// TwinCAT 3 PLC project mas516_PLC
// ProgramVersion: 3.1.4023.0
// libraries:
//   Tc2_Standard, * (Beckhoff Automation GmbH)
//   Tc2_System, * (Beckhoff Automation GmbH)
//   Tc3_Module, * (Beckhoff Automation GmbH)
//   VisuDialogs, * (System)
// project tree:
//   / GlobalTextList.TcGTLO, MAIN.TcPOU, PlcTask.TcTTO, Visualization Manager.TcVMO (not stored)
//   HMI/Function blocks/ FB_ModifyAutomaticControlSettings.TcPOU
//   HMI/ G_Hmi.TcGVL, Main.TcVIS
//   HMI/Struct/ ST_ModifyAutomaticControlSettings.TcDUT
//   HMI/Sub/ Cylinder.TcVIS, Winch.TcVIS
//   Inputs/Function blocks/ FB_AnalogInputScaling.TcPOU, FB_Encoder.TcPOU, FB_JoystickInputScaling.TcPOU, FB_FlowMeterInputScaling.TcPOU
//   Inputs/Functions/ F_DegToRad.TcPOU
//   Inputs/ G_Inputs.TcGVL, G_Sensors.TcGVL, P_Inputs.TcPOU
//   Inputs/Struct/ ST_AnalogInput.TcDUT, ST_JoystickInputScaling.TcDUT, ST_AnalogInputStatus.TcDUT, ST_AnalogInputScaling.TcDUT, ST_FlowMeterInputScaling.TcDUT
//   Machine Control/Function blocks/ FB_CylController.TcPOU, FB_AutomaticControl.TcPOU, FB_AutomaticControlWinch.TcPOU, FB_ClosedLoopControl.TcPOU, FB_FeedforwardWinch.TcPOU, FB_MotionReferenceGenerator_limit.TcPOU, FB_OpenLoopControl.TcPOU, FB_OpenLoopControlWinch.TcPOU, FB_ResetIntegralController.TcPOU, FB_ValveOutputGenerator.TcPOU, FB_AutomaticControl_old.TcPOU, FB_Clock.TcPOU, FB_ManualControl.TcPOU, FB_FeedForwardCyl.TcPOU, GVL_1247965427.TcGVL, FB_RampGen.TcPOU, WinchAngle.TcPOU (not stored)
//   Machine Control/ G_HeightCorrection.TcGVL, G_Parameters.TcGVL, G_Work.TcGVL, P_MachineControl.TcPOU
//   Machine Control/Struct/ ST_AutomaticControlSettings.TcDUT, ST_ClosedLoopControlSettings.TcDUT, ST_MotionReferenceGeneratorSettings.TcDUT, ST_OpenLoopControlSettings.TcDUT, ST_Parameters.TcDUT, ST_ValveOutputGeneratorSettings.TcDUT
//   Outputs/Function blocks/ FB_ValveOutput.TcPOU
//   Outputs/ G_Outputs.TcGVL, P_Outputs.TcPOU
//   Outputs/Struct/ ST_ValveDeadBand.TcDUT, ST_ValveOutput.TcDUT
// real-time tasks:
//   TASK PlcTask: cycle T#1ms, priority 20, ADS port 350
// I/O:
//   DEVICE Device 3 (EtherCAT), AmsNetId 128.39.200.184.4.1
//     Term 1 (EK1100) [EK1100 EtherCAT Coupler (2A E-Bus)]
//       DI (EL1008) [EL1008 8Ch. Dig. Input 24V, 3ms]
//       Term 3 (EL2008) [EL2008 8Ch. Dig. Output 24V, 0.5A]
//       Term 4 (EL3068) [EL3068 8Ch. Ana. Input 0-10V]
//       Term 5 (EL3068) [EL3068 8Ch. Ana. Input 0-10V]
//       Term 6 (EL3174) [EL3174 4Ch. Ana. Input +/-10V Diff., +/-20mA SingleEnded, 16 Bit]
//       Term 7 (EL3255) [EL3255 5Ch. potentiometer measurement with sensor supply]
//       Term 8 (EL4104) [EL4104 4Ch. Ana. Output 0-10V, 16bit]
//       Term 9 (EL6751) [EL6751 CANopen Master]
//       Term 11 (EL9011) [EL9011 End Terminal]
//     Box 10 (Fraba EtherCAT) [Absolute Rotary Encoder IXARC V01.05]
//   DEVICE Device 1 (EL6751), AmsNetId 128.39.200.184.2.1
// variable links:
//   mas516_PLC/mas516_PLC Instance <-> Device 3 (EtherCAT)/Box 10 (Fraba EtherCAT)
//     PlcTask Inputs/G_Inputs.nEncoderValue <-> Encoder/Position Value
//   mas516_PLC/mas516_PLC Instance <-> Device 3 (EtherCAT)/Term 1 (EK1100)/DI (EL1008)
//     PlcTask Inputs/G_Inputs.bAutoModeSelector <-> Channel 2/Input
//     PlcTask Inputs/G_Inputs.bJoystickEnable <-> Channel 5/Input
//     PlcTask Inputs/G_Inputs.bManualModeSelector <-> Channel 1/Input
//     PlcTask Inputs/G_Inputs.bStartButton <-> Channel 3/Input
//     PlcTask Inputs/G_Inputs.bStopButton <-> Channel 4/Input
//   mas516_PLC/mas516_PLC Instance <-> Device 3 (EtherCAT)/Term 1 (EK1100)/Term 3 (EL2008)
//     PlcTask Outputs/G_Outputs.bGreenLight <-> Channel 1/Output
//     PlcTask Outputs/G_Outputs.bRedLight <-> Channel 2/Output
//     PlcTask Outputs/G_Outputs.stCylValveOutput.bEnable <-> Channel 4/Output
//     PlcTask Outputs/G_Outputs.stWinchValveOutput.bEnable <-> Channel 3/Output
//   mas516_PLC/mas516_PLC Instance <-> Device 3 (EtherCAT)/Term 1 (EK1100)/Term 4 (EL3068)
//     PlcTask Inputs/G_Inputs.stPressureCyl_A_PistonSide.nValue <-> AI Standard Channel 4/Value
//     PlcTask Inputs/G_Inputs.stPressureCyl_A_PistonSide.stStatus <-> AI Standard Channel 4/Status
//     PlcTask Inputs/G_Inputs.stPressureCyl_B_RodSide.nValue <-> AI Standard Channel 3/Value
//     PlcTask Inputs/G_Inputs.stPressureCyl_B_RodSide.stStatus <-> AI Standard Channel 3/Status
//     PlcTask Inputs/G_Inputs.stPressureReturn.nValue <-> AI Standard Channel 2/Value
//     PlcTask Inputs/G_Inputs.stPressureReturn.stStatus <-> AI Standard Channel 2/Status
//     PlcTask Inputs/G_Inputs.stPressureSupply.nValue <-> AI Standard Channel 1/Value
//     PlcTask Inputs/G_Inputs.stPressureSupply.stStatus <-> AI Standard Channel 1/Status
//     PlcTask Inputs/G_Inputs.stPressureWinch_A1_Input.nValue <-> AI Standard Channel 5/Value
//     PlcTask Inputs/G_Inputs.stPressureWinch_A1_Input.stStatus <-> AI Standard Channel 5/Status
//     PlcTask Inputs/G_Inputs.stPressureWinch_A_Input.nValue <-> AI Standard Channel 7/Value
//     PlcTask Inputs/G_Inputs.stPressureWinch_A_Input.stStatus <-> AI Standard Channel 7/Status
//     PlcTask Inputs/G_Inputs.stPressureWinch_B1_Output.nValue <-> AI Standard Channel 6/Value
//     PlcTask Inputs/G_Inputs.stPressureWinch_B1_Output.stStatus <-> AI Standard Channel 6/Status
//     PlcTask Inputs/G_Inputs.stPressureWinch_B_Output.nValue <-> AI Standard Channel 8/Value
//     PlcTask Inputs/G_Inputs.stPressureWinch_B_Output.stStatus <-> AI Standard Channel 8/Status
//   mas516_PLC/mas516_PLC Instance <-> Device 3 (EtherCAT)/Term 1 (EK1100)/Term 5 (EL3068)
//     PlcTask Inputs/G_Inputs.stPressureWinchDrain.nValue <-> AI Standard Channel 1/Value
//     PlcTask Inputs/G_Inputs.stPressureWinchDrain.stStatus <-> AI Standard Channel 1/Status
//   mas516_PLC/mas516_PLC Instance <-> Device 3 (EtherCAT)/Term 1 (EK1100)/Term 6 (EL3174)
//     PlcTask Inputs/G_Inputs.stFlowWinch.nValue <-> AI Standard Channel 1/Value
//     PlcTask Inputs/G_Inputs.stFlowWinch.stStatus <-> AI Standard Channel 1/Status
//   mas516_PLC/mas516_PLC Instance <-> Device 3 (EtherCAT)/Term 1 (EK1100)/Term 7 (EL3255)
//     PlcTask Inputs/G_Inputs.stJoyX.nValue <-> AI Standard Channel 2/Value
//     PlcTask Inputs/G_Inputs.stJoyX.stStatus <-> AI Standard Channel 2/Status
//     PlcTask Inputs/G_Inputs.stJoyY.nValue <-> AI Standard Channel 3/Value
//     PlcTask Inputs/G_Inputs.stJoyY.stStatus <-> AI Standard Channel 3/Status
//     PlcTask Inputs/G_Inputs.stPositionCylPiston.nValue <-> AI Standard Channel 1/Value
//     PlcTask Inputs/G_Inputs.stPositionCylPiston.stStatus <-> AI Standard Channel 1/Status
//   mas516_PLC/mas516_PLC Instance <-> Device 3 (EtherCAT)/Term 1 (EK1100)/Term 8 (EL4104)
//     PlcTask Outputs/G_Outputs.stCylValveOutput.nValveOutput <-> AO Output Channel 2/Analog output
//     PlcTask Outputs/G_Outputs.stWinchValveOutput.nValveOutput <-> AO Output Channel 1/Analog output

CONFIGURATION mas516_PLC
    RESOURCE PLC ON TwinCAT3
        TASK PlcTask(INTERVAL := T#1ms, PRIORITY := 20);
        PROGRAM MAIN WITH PlcTask : MAIN;
    END_RESOURCE
END_CONFIGURATION

// ---- HMI/Struct/ST_ModifyAutomaticControlSettings.TcDUT
TYPE ST_ModifyAutomaticControlSettings :
STRUCT
	bSetNewMaxFlowCapacity		: BOOL;
	fNewMaxFlowCapacity 		: LREAL;
	bSetNewProportionalGain 	: BOOL;
	bSetNewIntegralGain 		: BOOL;
	fNewProportionalGain 		: LREAL;
	fNewIntegralGain 			: LREAL;
	bSetNewMaxPositionError 	: BOOL;
	fNewMaxPositionError		: LREAL;
END_STRUCT
END_TYPE

// ---- Inputs/Struct/ST_AnalogInput.TcDUT
TYPE ST_AnalogInput :
STRUCT
	stStatus 	AT %I* : ST_AnalogInputStatus;
	nValue		AT %I* : INT;	
END_STRUCT
END_TYPE

// ---- Inputs/Struct/ST_JoystickInputScaling.TcDUT
TYPE ST_JoystickInputScaling :
STRUCT
	fMaxInputValue			: LREAL;	// tunable max input value
	fMinInputValue 			: LREAL;	// tunable min input value
	fNeutralInputValue  	: LREAL;	// tunable neutral input value
	fNeutralDeadband		: LREAL;	// tunable dead_band value
	fMaxOutputValue  		: LREAL;	// normalized max output value
	fMinOutputValue  		: LREAL;	// normalized min output value
	fNeutralOutputValue  	: LREAL;	// normalized neutral output value
END_STRUCT
END_TYPE

// ---- Inputs/Struct/ST_AnalogInputStatus.TcDUT
TYPE ST_AnalogInputStatus :
STRUCT
	Underrange 		: BIT; // 0.0
	Overrange 		: BIT; // 0.1
	Limit_1_0 		: BIT; // 0.2
	Limit_1_1 		: BIT; // 0.3
	Limit_2_0 		: BIT; // 0.4
	Limit_2_1 		: BIT; // 0.5
	Error 			: BIT; // 0.6
	Reserved_0_7	: BIT; // 0.7
	Reserved_1_0 	: BIT; // 1.0
	Reserved_1_1 	: BIT; // 1.1
	Reserved_1_2 	: BIT; // 1.2
	Reserved_1_3 	: BIT; // 1.3
	Reserved_1_4 	: BIT; // 1.4
	Reserved_1_5 	: BIT; // 1.5
	TxPDO_State 	: BIT; // 1.6
	TxPDO_Toggle 	: BIT; // 1.7	
END_STRUCT
END_TYPE

// ---- Inputs/Struct/ST_AnalogInputScaling.TcDUT
TYPE ST_AnalogInputScaling :
STRUCT
	fMaxInputValue 			: LREAL;	// tunable max input value 
	fMinInputValue			: LREAL;	// tunable min input value  
	fMaxOutputValue  		: LREAL;	// max sensor output value
	fMinOutputValue  		: LREAL;	// min sensor output value	
END_STRUCT
END_TYPE

// ---- Inputs/Struct/ST_FlowMeterInputScaling.TcDUT
TYPE ST_FlowMeterInputScaling :
STRUCT
	fMaxInputValue			: LREAL;	// tunable max input value
	fMinInputValue 			: LREAL;	// tunable min input value
	fNeutralInputValue  	: LREAL;	// tunable neutral input value
	fNeutralDeadband		: LREAL;	// tunable dead_band value
	fMaxOutputValue  		: LREAL;	// normalized max output value
	fMinOutputValue  		: LREAL;	// normalized min output value
	fNeutralOutputValue  	: LREAL;	// normalized neutral output value
END_STRUCT
END_TYPE

// ---- Machine Control/Struct/ST_AutomaticControlSettings.TcDUT
TYPE ST_AutomaticControlSettings :
STRUCT
	bEnableVelocityFeedForwardControl	: BOOL;
	bEnableClosedLoopPositionControl	: BOOL;
	bEnableIntegralController 			: BOOL;
	bEnableActiveDamping 				: BOOL;	
END_STRUCT
END_TYPE

// ---- Machine Control/Struct/ST_ClosedLoopControlSettings.TcDUT
TYPE ST_ClosedLoopControlSettings :
STRUCT
	fMaxPositionError 					: LREAL;
	fProportionalGain 					: LREAL;
	fIntegralGain 						: LREAL;
END_STRUCT
END_TYPE

// ---- Machine Control/Struct/ST_MotionReferenceGeneratorSettings.TcDUT
TYPE ST_MotionReferenceGeneratorSettings :
STRUCT
	fStartPosition_m		: LREAL := 0.0;
	fStartVelocity_m		: LREAL	:= 0.0;
	fPositionSetpoint_ms	: LREAL := 0.25;
	fVelocitySetpoint_m		: LREAL := 0.025;
	fMaxPosition 			: LREAL := 0.7;
	fMinPosition 			: LREAL := 0.0;
	fMaxVelocity 			: LREAL := 0.05;
	fTimeBeforeStarting_s	: LREAL := 3.0;
	fRampTime_s				: LREAL := 1.0;
	fHoldPositionTime_s		: LREAL := 5.0;
END_STRUCT
END_TYPE

// ---- Machine Control/Struct/ST_OpenLoopControlSettings.TcDUT
TYPE ST_OpenLoopControlSettings :
STRUCT
	fBoreArea 			: LREAL;
	fAnnulusArea 		: LREAL;
	fMaxFlowCapacity 	: LREAL; //[l/min]
END_STRUCT
END_TYPE

// ---- Machine Control/Struct/ST_Parameters.TcDUT
TYPE ST_Parameters :
STRUCT
	fCyclicTime 					: LREAL := 0.001; // [s]
	fMaxCylVelocityLimit 			: LREAL := 0.005; // [m/s]
	fMaxWinchVelocityLimit 			: LREAL := 0.005; // [rad/s]
	bDeadBandCompOn 				: BOOL := TRUE;
	stWinchValveDeadBand 			: ST_ValveDeadBand := (fPosMax := 29490.0, fPosMin := 20950.0, fNegMin := 18250.0, fNegMax := 9830.0);
	stCylValveDeadBand 				: ST_ValveDeadBand := (fPosMax := 29490.0, fPosMin := 20950.0, fNegMin := 18250.0, fNegMax := 9830.0);
	stPressureSensorScaling400bar 	: ST_AnalogInputScaling := (fMaxInputValue := 32767.0, fMinInputValue := 0.0, fMaxOutputValue := 400.0, fMinOutputValue := 0.0);
	stPressureSensorScaling40bar 	: ST_AnalogInputScaling := (fMaxInputValue := 32767.0, fMinInputValue := 0.0, fMaxOutputValue := 40.0, fMinOutputValue := 0.0);
	stJoystickInputScalingX 		: ST_JoystickInputScaling := (fMaxInputValue := 20509.0, fMinInputValue := 11787.0, fNeutralInputValue := 16175, fNeutralDeadband := 50.0, fMaxOutputValue := 1.0, fMinOutputValue := -1.0, fNeutralOutputValue := 0.0);
	stCylPistonPositionScaling 		: ST_AnalogInputScaling := (fMaxInputValue := 32295.0, fMinInputValue := 229.0, fMaxOutputValue := 0.5, fMinOutputValue := 0.0);
	stFlowMeterInputScaling 		: ST_FlowMeterInputScaling := (fMaxInputValue := 32295.0, fMinInputValue := 0.0, fNeutralInputValue := 15450, fNeutralDeadband := 50.0, fMaxOutputValue := 150.0, fMinOutputValue := -150.0, fNeutralOutputValue := 0.0);
	stJoystickInputScalingY 		: ST_JoystickInputScaling := (fMaxInputValue := 20504.0, fMinInputValue := 12160.0, fNeutralInputValue := 16640, fNeutralDeadband := 50.0, fMaxOutputValue := 1.0, fMinOutputValue := -1.0, fNeutralOutputValue := 0.0);
	fEncoderOffset 					: LREAL := 17574.8; // Encoder value at zero (Cylinder out / second layaer)
	fWinchDrumScaling				: LREAL := 0.000744309; //  (empirical value - combined drum diameter and gearing)
	fWinchSpeedReducerGain 			: LREAL := 0.2;
	fCylSpeedReducerGain 			: LREAL := 0.2;
	fDisplacment_cc 				: LREAL := 32;
	stWinchValveOutputGeneratorSettings  	: ST_ValveOutputGeneratorSettings := (fInitialValveOpening := 0.0, fValveOpeningSetPoint := 0.2, fTimeBeforeStarting_s := 3.0, fRampTime_s := 1.0, fHoldTime_s := 1.0, fWaitTime_s := 5.0);
	stCylValveOutputGeneratorSettings  		: ST_ValveOutputGeneratorSettings := (fInitialValveOpening := 0.0, fValveOpeningSetPoint := 0.2, fTimeBeforeStarting_s := 3.0, fRampTime_s := 1.0, fHoldTime_s := 1.0, fWaitTime_s := 5.0);
	stOpenLoopControlSettingsWinch 			: ST_OpenLoopControlSettings := (fBoreArea := 0.0, fAnnulusArea := 0.0, fMaxFlowCapacity := 60.0);
	stClosedLoopControlSettingsWinch 		: ST_ClosedLoopControlSettings := (fMaxPositionError := 2E-3, fProportionalGain := 9.7, fIntegralGain := 6.5);
	stOpenLoopControlSettingsCylinder 		: ST_OpenLoopControlSettings := (fBoreArea := 0.0033183, fAnnulusArea := 0.0023562, fMaxFlowCapacity := 75.0);
	stClosedLoopControlSettingsCylinder 	: ST_ClosedLoopControlSettings := (fMaxPositionError := 2E-3, fProportionalGain := 14.6, fIntegralGain := 9.75);	
END_STRUCT
END_TYPE

// ---- Machine Control/Struct/ST_ValveOutputGeneratorSettings.TcDUT
TYPE ST_ValveOutputGeneratorSettings :
STRUCT
	fInitialValveOpening	:	LREAL;
	fValveOpeningSetPoint	:	LREAL;
	fTimeBeforeStarting_s	:	LREAL;
	fRampTime_s				:	LREAL;
	fHoldTime_s				:	LREAL;
	fWaitTime_s				:	LREAL;
END_STRUCT
END_TYPE

// ---- Outputs/Struct/ST_ValveDeadBand.TcDUT
TYPE ST_ValveDeadBand :
STRUCT
	fPosMax	: LREAL; // Positive min value [19660..29490]
	fPosMin	: LREAL; // Positive max value [19660..29490]
	fNegMin : LREAL; // Negative max value [9830..19660]
	fNegMax	: LREAL; // Negative min value [9830..19660]
END_STRUCT
END_TYPE

// ---- Outputs/Struct/ST_ValveOutput.TcDUT
TYPE ST_ValveOutput :
STRUCT
	bEnable					AT %Q* : BOOL := 0;
	nValveOutput 			AT %Q* : INT := 19660;
END_STRUCT
END_TYPE

// ---- HMI/G_Hmi.TcGVL
{attribute 'qualified_only'}
VAR_GLOBAL
	bWinchEnable	: BOOL;
	bCylEnable 		: BOOL;
	stAutomaticControlSettingsWinch 			: ST_AutomaticControlSettings;
	stMotionReferenceGeneratorSettingsWinch  	: ST_MotionReferenceGeneratorSettings;
	stAutomaticControlSettingsCylinder 			: ST_AutomaticControlSettings;
	stMotionReferenceGeneratorSettingsCylinder  : ST_MotionReferenceGeneratorSettings;
	stModifyAutomaticControlSettingsWinch 		: ST_ModifyAutomaticControlSettings;
	stModifyAutomaticControlSettingsCylinder 	: ST_ModifyAutomaticControlSettings;
END_VAR

// ---- Inputs/G_Inputs.TcGVL
{attribute 'qualified_only'}
VAR_GLOBAL
	bManualModeSelector			AT %I* : BOOL;
	bAutoModeSelector			AT %I* : BOOL;
	bStartButton				AT %I* : BOOL;
	bStopButton					AT %I* : BOOL;
	bJoystickEnable				AT %I* : BOOL;
	
	// Analog Inputs 1
	stJoyX 						: ST_AnalogInput;
	stJoyY						: ST_AnalogInput;
	stPositionCylPiston 		: ST_AnalogInput;
	nEncoderValue 				AT %I* : UDINT;
	
	// Analog Inputs 2
	// HPU Interface
	stPressureSupply 			: ST_AnalogInput;
	stPressureReturn 			: ST_AnalogInput;
	// Cylinder
	stPressureCyl_A_PistonSide 	: ST_AnalogInput;
	stPressureCyl_B_RodSide		: ST_AnalogInput;
	// Winch
	stPressureWinch_A_Input 	: ST_AnalogInput;
	stPressureWinch_A1_Input 	: ST_AnalogInput;
	stPressureWinch_B_Output	: ST_AnalogInput;
	stPressureWinch_B1_Output	: ST_AnalogInput;
	stPressureWinchDrain		: ST_AnalogInput;
	
	// Analog Inputs 3 (Multi)
	stFlowWinch					: ST_AnalogInput;
END_VAR

// ---- Inputs/G_Sensors.TcGVL
{attribute 'qualified_only'}
VAR_GLOBAL
	fJoystickNormalizedY 		: LREAL;
	fJoystickNormalizedX 		: LREAL;
	fPositionCylPiston  		: LREAL;
	// HPU Interface
	fPressureSupply 			: LREAL;
	fPressureReturn 			: LREAL;
	// Cylinder
	fPressureCyl_A_PistonSide 	: LREAL;
	fPressureCyl_B_RodSide		: LREAL;
	// Winch
	fPressureWinch_A_Input 		: LREAL;
	fPressureWinch_A1_Side 		: LREAL;
	fPressureWinch_B_Output		: LREAL;
	fPressureWinch_B1_Output	: LREAL;
	fPressureWinchDrain			: LREAL;
	fWinchEncoderPosition 		: LREAL;
	fWinchWirePosition 			: LREAL;
	fWinchFlow 					: LREAL;	// [L/min]
END_VAR

// ---- Machine Control/Function blocks/GVL_1247965427.TcGVL
VAR_GLOBAL CONSTANT
	SS_INITIALIZE: SINT := 0;
	SS_STEP: SINT := 1;
END_VAR

// ---- Machine Control/G_HeightCorrection.TcGVL
{attribute 'qualified_only'}
VAR_GLOBAL
	xCorrectHeight : BOOL;
	rZeroOffset : REAL;
	rActual: REAL;
	rDesiredHeight: REAL;
END_VAR

// ---- Machine Control/G_Parameters.TcGVL
{attribute 'qualified_only'}
VAR_GLOBAL
	stParam : ST_Parameters;
END_VAR

// ---- Machine Control/G_Work.TcGVL
{attribute 'qualified_only'}
VAR_GLOBAL
	bManualMode 			: BOOL;
	bAutoMode 				: BOOL;
	bWinchEnable 			: BOOL;
	bCylEnable 				: BOOL;
	fWinchControlInput 		: LREAL;
	fWinchTime				: LREAL;
	fCylControlInput 		: LREAL;
	fCylTime				: LREAL;
	fVelRefWinch 			: LREAL;
	fPosRefWinch 			: LREAL;
	fControlSignWinch		: LREAL;
	fVelRefCyl 				: LREAL;
	fPosRefCyl 				: LREAL;
	fControlSignCyl			: LREAL;
	fPositionErrorWinch_mm 	: LREAL;
	fPositionErrorCylinder_mm : LREAL;
END_VAR

// ---- Outputs/G_Outputs.TcGVL
{attribute 'qualified_only'}
VAR_GLOBAL
	// PLC Rack
	
	// RIO Rack
	// Digital Outputs
	bGreenLight 			AT %Q* : BOOL;
	bRedLight 				AT %Q* : BOOL;
	// Analog Outputs
	stWinchValveOutput 		: ST_ValveOutput;
	stCylValveOutput 		: ST_ValveOutput;
END_VAR

// ---- MAIN.TcPOU
PROGRAM MAIN
VAR
END_VAR

P_Inputs();
P_MachineControl();
P_Outputs();

END_PROGRAM

// ---- Inputs/P_Inputs.TcPOU
PROGRAM P_Inputs
VAR
	fbJoystickWinch 				: FB_JoystickInputScaling;
	fbJoystickCyl 					: FB_JoystickInputScaling;
	fbWinchPosition 				: FB_Encoder;
	fbCylPistonPosition 			: FB_AnalogInputScaling;
	fbPressureSupply 				: FB_AnalogInputScaling;
	fbPressureReturn 				: FB_AnalogInputScaling;
	fbPressureCyl_A_PistonSide 		: FB_AnalogInputScaling;
	fbPressureCyl_B_RodSide			: FB_AnalogInputScaling;
	fbPressureWinch_A_Input 		: FB_AnalogInputScaling;
	fbPressureWinch_A1_Input 		: FB_AnalogInputScaling;
	fbPressureWinch_B_Output		: FB_AnalogInputScaling;
	fbPressureWinch_B1_Output		: FB_AnalogInputScaling;
	fbPressureWinchDrain			: FB_AnalogInputScaling;
	fbFlowWinch						: FB_FlowMeterInputScaling;
	
	
	
END_VAR

fbJoystickWinch(
	bEnable := G_Work.bManualMode,
	nRawInput := G_Inputs.stJoyY.nValue,
	stJoystickInputScaling := G_Parameters.stParam.stJoystickInputScalingY,
	fNormalizedOutput => G_Sensors.fJoystickNormalizedY
);

fbJoystickCyl(
	bEnable := G_Work.bManualMode,
	nRawInput := G_Inputs.stJoyX.nValue,
	stJoystickInputScaling := G_Parameters.stParam.stJoystickInputScalingX,
	fNormalizedOutput => G_Sensors.fJoystickNormalizedX
);

fbWinchPosition (
nRawInput := G_Inputs.nEncoderValue, 
fPosition => G_Sensors.fWinchEncoderPosition,
);

G_Sensors.fWinchWirePosition := fbWinchPosition.fPosition*G_Parameters.stParam.fWinchDrumScaling;

fbCylPistonPosition(
	nRawInput := G_Inputs.stPositionCylPiston.nValue,
	stAnalogInputScaling := G_Parameters.stParam.stCylPistonPositionScaling,
	fOutput => G_Sensors.fPositionCylPiston
);

fbPressureSupply(
	nRawInput := G_Inputs.stPressureSupply.nValue,
	stAnalogInputScaling := G_Parameters.stParam.stPressureSensorScaling400bar,
	fOutput => G_Sensors.fPressureSupply
);

fbPressureReturn(
	nRawInput := G_Inputs.stPressureReturn.nValue,
	stAnalogInputScaling := G_Parameters.stParam.stPressureSensorScaling40bar,
	fOutput => G_Sensors.fPressureReturn
);

fbPressureCyl_A_PistonSide(
	nRawInput := G_Inputs.stPressureCyl_A_PistonSide.nValue,
	stAnalogInputScaling := G_Parameters.stParam.stPressureSensorScaling400bar,
	fOutput => G_Sensors.fPressureCyl_A_PistonSide
);

fbPressureCyl_B_RodSide(
	nRawInput := G_Inputs.stPressureCyl_B_RodSide.nValue,
	stAnalogInputScaling := G_Parameters.stParam.stPressureSensorScaling400bar,
	fOutput => G_Sensors.fPressureCyl_B_RodSide
);

fbPressureWinch_A_Input(
	nRawInput := G_Inputs.stPressureWinch_A_Input.nValue,
	stAnalogInputScaling := G_Parameters.stParam.stPressureSensorScaling400bar,
	fOutput => G_Sensors.fPressureWinch_A_Input
);

fbPressureWinch_A1_Input(
	nRawInput := G_Inputs.stPressureWinch_A1_Input.nValue,
	stAnalogInputScaling := G_Parameters.stParam.stPressureSensorScaling400bar,
	fOutput => G_Sensors.fPressureWinch_A1_Side
);

fbPressureWinch_B_Output(
	nRawInput := G_Inputs.stPressureWinch_B_Output.nValue,
	stAnalogInputScaling := G_Parameters.stParam.stPressureSensorScaling400bar,
	fOutput => G_Sensors.fPressureWinch_B_Output
);

fbPressureWinch_B1_Output(
	nRawInput := G_Inputs.stPressureWinch_B1_Output.nValue,
	stAnalogInputScaling := G_Parameters.stParam.stPressureSensorScaling400bar,
	fOutput => G_Sensors.fPressureWinch_B1_Output
);

fbPressureWinchDrain(
	nRawInput := G_Inputs.stPressureWinchDrain.nValue,
	stAnalogInputScaling := G_Parameters.stParam.stPressureSensorScaling40bar,
	fOutput => G_Sensors.fPressureWinchDrain
);

fbFlowWinch(
	nRawInput := G_Inputs.stFlowWinch.nValue,
	stFlowMeterInputScaling := G_Parameters.stParam.stFlowMeterInputScaling,
	fNormalizedOutput => G_Sensors.fWinchFlow
);

END_PROGRAM

// ---- Inputs/Function blocks/FB_JoystickInputScaling.TcPOU
FUNCTION_BLOCK FB_JoystickInputScaling
VAR_INPUT
	bEnable 				: BOOL;
	nRawInput 				: INT;
	stJoystickInputScaling  : ST_JoystickInputScaling;
END_VAR
VAR_OUTPUT
	fNormalizedOutput 		: LREAL;
END_VAR
VAR
	fRawInput 				: LREAL;
	fTempInput 				: LREAL;
	fTempOutput 			: LREAL;
END_VAR

fRawInput := INT_TO_LREAL(nRawInput);

fTempInput := fRawInput - stJoystickInputScaling.fNeutralInputValue;

IF fTempInput > stJoystickInputScaling.fNeutralDeadband THEN
	fTempOutput := fTempInput/(stJoystickInputScaling.fMaxInputValue - stJoystickInputScaling.fNeutralInputValue);
ELSIF fTempInput < -stJoystickInputScaling.fNeutralDeadband THEN	
	fTempOutput := fTempInput/(stJoystickInputScaling.fNeutralInputValue - stJoystickInputScaling.fMinInputValue);
ELSE
	fTempOutput := 0.0;
END_IF

IF NOT(bEnable) THEN
	fNormalizedOutput := 0.0;
ELSE
	fNormalizedOutput := LIMIT(stJoystickInputScaling.fMinOutputValue, fTempOutput, stJoystickInputScaling.fMaxOutputValue);
END_IF

END_FUNCTION_BLOCK

// ---- Inputs/Function blocks/FB_Encoder.TcPOU
FUNCTION_BLOCK FB_Encoder
VAR_INPUT
	nRawInput : UDINT;
	stParam 		: ST_Parameters; 
END_VAR
VAR_OUTPUT
	fPosition 		: LREAL;
END_VAR
VAR PERSISTENT
	nRounds			: DINT;
	nRawLast 		: DINT;
END_VAR	
VAR
	nInput 		: DINT;
	nTempInputDiff	: DINT;
	nCount 			: DINT;
	nMaxValue30bit 	: DINT :=  1073741823; // 2^30 - 1	
	nThreshold30bit	: DINT := nMaxValue30bit/2;
	fScale16bit		: LREAL := 360.0/65535.0; // 360deg/(2^16 - 1)
	fTempPosition   : LREAL;
END_VAR

// Convert to DINT (same as const values)
nInput := UDINT_TO_DINT(nRawInput);

// Define Encoder Rounds
nTempInputDiff := nInput - nRawLast;
IF (nTempInputDiff > nThreshold30bit) THEN
	nRounds := nRounds - 1;
END_IF

IF (nTempInputDiff < -nThreshold30bit) THEN
	nRounds := nRounds + 1;
END_IF

// Count Encoder Rounds
nCount := nInput + nRounds*nMaxValue30bit;

//Position Output
fPosition := DINT_TO_LREAL(nCount)*fScale16bit - stParam.fEncoderOffset; // [deg]

END_FUNCTION_BLOCK

// ---- Inputs/Function blocks/FB_AnalogInputScaling.TcPOU
FUNCTION_BLOCK FB_AnalogInputScaling
VAR_INPUT
	nRawInput 				: INT;
	stAnalogInputScaling    : ST_AnalogInputScaling;
END_VAR
VAR_OUTPUT
	fOutput 				: LREAL;
END_VAR
VAR
	fRawInput 				: LREAL;
	fNormalizedInput		: LREAL;
END_VAR

fRawInput := INT_TO_LREAL(nRawInput);

fNormalizedInput := (fRawInput - stAnalogInputScaling.fMinInputValue) / (stAnalogInputScaling.fMaxInputValue - stAnalogInputScaling.fMinInputValue);

fOutput := LIMIT(stAnalogInputScaling.fMinOutputValue, stAnalogInputScaling.fMinOutputValue + fNormalizedInput*(stAnalogInputScaling.fMaxOutputValue - stAnalogInputScaling.fMinOutputValue), stAnalogInputScaling.fMaxOutputValue);

END_FUNCTION_BLOCK

// ---- Inputs/Function blocks/FB_FlowMeterInputScaling.TcPOU
FUNCTION_BLOCK FB_FlowMeterInputScaling
VAR_INPUT
	nRawInput 				: INT;
	stFlowMeterInputScaling  : ST_FlowMeterInputScaling;
END_VAR
VAR_OUTPUT
	fNormalizedOutput 		: LREAL;
END_VAR
VAR
	fRawInput 				: LREAL;
	fTempInput 				: LREAL;
	fTempOutput 			: LREAL;
END_VAR

fRawInput := INT_TO_LREAL(nRawInput);

fTempInput := fRawInput - stFlowMeterInputScaling.fNeutralInputValue;

IF fTempInput > stFlowMeterInputScaling.fNeutralDeadband THEN
	fTempOutput := fTempInput/(stFlowMeterInputScaling.fMaxInputValue - stFlowMeterInputScaling.fNeutralInputValue);
ELSIF fTempInput < -stFlowMeterInputScaling.fNeutralDeadband THEN	
	fTempOutput := fTempInput/(stFlowMeterInputScaling.fNeutralInputValue - stFlowMeterInputScaling.fMinInputValue);
ELSE
	fTempOutput := 0.0;
END_IF

fNormalizedOutput := LIMIT(stFlowMeterInputScaling.fMinOutputValue, fTempOutput*150.0, stFlowMeterInputScaling.fMaxOutputValue);

END_FUNCTION_BLOCK

// ---- Machine Control/P_MachineControl.TcPOU
PROGRAM P_MachineControl
VAR
	fbManualControlWinch 		: FB_ManualControl;
	fbManualControlCyl	 		: FB_ManualControl;
	//fbAutomaticControlWinch 	: FB_AutomaticControl_old;
	//fbAutomaticControlCyl	 	: FB_AutomaticControl_old;
	fWinchControlSignalManual 			: LREAL;
	fCylControlSignalManual 			: LREAL;
	fWinchControlSignalAuto 			: LREAL;
	fCylControlSignalAuto				: LREAL;
	fbAutomaticControlWinch 	:	FB_AutomaticControlWinch;
	fbAutomaticControlCylinder 		:	FB_AutomaticControl;
	fbModifyAutomaticControlSettingsWinch : FB_ModifyAutomaticControlSettings;
	fbModifyAutomaticControlSettingsCylinder : FB_ModifyAutomaticControlSettings;
END_VAR

G_Work.bManualMode := G_Inputs.bManualModeSelector;
G_Work.bAutoMode := G_Inputs.bAutoModeSelector;

G_Work.bWinchEnable := (G_Hmi.bWinchEnable AND G_Inputs.bJoystickEnable);
G_Work.bCylEnable :=  (G_Hmi.bCylEnable AND G_Inputs.bJoystickEnable);

fbManualControlWinch(
	bEnable := G_Work.bManualMode AND G_Work.bWinchEnable,
	fInput := G_Sensors.fJoystickNormalizedY*-G_Parameters.stParam.fWinchSpeedReducerGain,
	fControlRefSignal => fWinchControlSignalManual
);

fbManualControlCyl(
	bEnable := G_Work.bManualMode AND G_Work.bCylEnable,
	fInput := G_Sensors.fJoystickNormalizedX*G_Parameters.stParam.fCylSpeedReducerGain,
	fControlRefSignal => fCylControlSignalManual
);

//fbAutomaticControlWinch(
//	bEnable := G_Work.bAutoMode AND G_Hmi.bWinchEnable,
//	bStartMotion := G_Inputs.bStartButton,
//	bStopMotion := G_Inputs.bStopButton,
//	stValveOutputGeneratorSettings := G_Parameters.stWinchValveOutputGeneratorSettings,
//	fNormalizedValveOpeningRefSignal => fWinchControlSignalAuto,
//	fTime => G_Work.fWinchTime
//);

//fbAutomaticControlCyl(
//	bEnable := G_Work.bAutoMode AND G_Hmi.bCylEnable,
//	bStartMotion := G_Inputs.bStartButton,
//	bStopMotion := G_Inputs.bStopButton,
//	stValveOutputGeneratorSettings := G_Parameters.stCylValveOutputGeneratorSettings,
//	fNormalizedValveOpeningRefSignal => fCylControlSignalAuto,
//	fTime => G_Work.fCylTime
//);

fbModifyAutomaticControlSettingsWinch(
	stParamOpenLoopControllSettings := G_Parameters.stParam.stOpenLoopControlSettingsWinch,
	stParamClosedLoopControllSettings := G_Parameters.stParam.stClosedLoopControlSettingsWinch,	
	stModify := G_Hmi.stModifyAutomaticControlSettingsWinch
);

fbAutomaticControlWinch(
	bEnable := G_Work.bAutoMode AND G_Hmi.bWinchEnable,
	bStartMotion := G_Inputs.bStartButton,
	bStopMotion := G_Inputs.bStopButton,
	stMotionReferenceGeneratorSettings := G_Hmi.stMotionReferenceGeneratorSettingsWinch,
	stAutomaticControlSettings := G_Hmi.stAutomaticControlSettingsWinch,
	stClosedLoopControlSettings := G_Parameters.stParam.stClosedLoopControlSettingsWinch,
	stOpenLoopControlSettings := G_Parameters.stParam.stOpenLoopControlSettingsWinch,
	stParam := G_Parameters.stParam,
	fPositionFeedback := G_Sensors.fWinchWirePosition,
	fVelocityReference_ms => G_Work.fVelRefWinch,
	fPositionReference_m => G_Work.fPosRefWinch,
	fTime => G_Work.fWinchTime,
	fPositionError_mm => G_Work.fPositionErrorWinch_mm,
	fControlOutputNormalized => G_Work.fControlSignWinch
);


fbModifyAutomaticControlSettingsCylinder(
	stParamOpenLoopControllSettings := G_Parameters.stParam.stOpenLoopControlSettingsCylinder,
	stParamClosedLoopControllSettings := G_Parameters.stParam.stClosedLoopControlSettingsCylinder,	
	stModify := G_Hmi.stModifyAutomaticControlSettingsCylinder
);

fbAutomaticControlCylinder(
	bEnable := G_Work.bAutoMode AND G_Hmi.bCylEnable,
	bStartMotion := G_Inputs.bStartButton,
	bStopMotion := G_Inputs.bStopButton,
	stMotionReferenceGeneratorSettings := G_Hmi.stMotionReferenceGeneratorSettingsCylinder,
	stAutomaticControlSettings := G_Hmi.stAutomaticControlSettingsCylinder,
	stClosedLoopControlSettings := G_Parameters.stParam.stClosedLoopControlSettingsCylinder,
	stOpenLoopControlSettings := G_Parameters.stParam.stOpenLoopControlSettingsCylinder,
	stParam := G_Parameters.stParam,
	fPositionFeedback := G_Sensors.fPositionCylPiston,
	fVelocityReference_ms => G_Work.fVelRefCyl,
	fPositionReference_m => G_Work.fPosRefCyl,
	fTime => G_Work.fCylTime,
	fPositionError_mm => G_Work.fPositionErrorCylinder_mm,
	fControlOutputNormalized => G_Work.fControlSignCyl
);

IF G_Work.bManualMode THEN
	G_Work.fWinchControlInput := fWinchControlSignalManual;
	G_Work.fCylControlInput := fCylControlSignalManual;
ELSIF G_Work.bAutoMode THEN
	G_Work.fWinchControlInput := G_Work.fControlSignWinch;
	G_Work.fCylControlInput := -G_Work.fControlSignCyl;
ELSE
	G_Work.fWinchControlInput := 0.0; 
	G_Work.fCylControlInput := 0.0;
END_IF

END_PROGRAM

// ---- Machine Control/Function blocks/FB_ManualControl.TcPOU
FUNCTION_BLOCK FB_ManualControl
VAR_INPUT
	bEnable 			: BOOL;
	fInput 				: LREAL;
END_VAR
VAR_OUTPUT
	fControlRefSignal	: LREAL;
END_VAR
VAR
END_VAR

IF NOT(bEnable) THEN
	fControlRefSignal := 0.0;
ELSE
	fControlRefSignal := fInput;
END_IF

END_FUNCTION_BLOCK

// ---- Machine Control/Function blocks/FB_AutomaticControlWinch.TcPOU
FUNCTION_BLOCK FB_AutomaticControlWinch
VAR_INPUT
	bEnable 							: BOOL;
	bStartMotion 						: BOOL;
	bStopMotion 						: BOOL;
	stMotionReferenceGeneratorSettings  : ST_MotionReferenceGeneratorSettings;
	stAutomaticControlSettings 			: ST_AutomaticControlSettings;
	stClosedLoopControlSettings 		: ST_ClosedLoopControlSettings;
	stOpenLoopControlSettings			: ST_OpenLoopControlSettings;
	stParam 							: ST_Parameters; 
	fPositionFeedback					: LREAL;
	rWinchPosRad						: REAL;
	fbHeightCalc						: WinchAngle;
	rActPos								: REAL;
	rSetPos								: REAL;
END_VAR
VAR_OUTPUT
	fTime : LREAL;
	fVelocityReference_ms : LREAL;
	fPositionReference_m : LREAL;
	fControlOutputNormalized : LREAL;
	fPositionError_mm : LREAL;
END_VAR
VAR
	fbClock : FB_Clock;	
	fbMotionReferenceGenerator 		: FB_MotionReferenceGenerator_limit;	
	fbVelocityFeedForwardControl 	: FB_FeedForwardWinch;
	fbResetIntegralController 		: FB_ResetIntegralController; 
	fbClosedLoopPositionControl 	: FB_CylController;
END_VAR

fbClock(
	bEnable := bEnable,
	bStart := bStartMotion,
	bStop := bStopMotion,
	fCycleTime := G_Parameters.stParam.fCyclicTime
);

fbMotionReferenceGenerator(
	bEnable := bEnable,
	stMotionReferenceGeneratorSettings := stMotionReferenceGeneratorSettings,
	fClock_s := fbClock.fTime
);

fbVelocityFeedForwardControl(
	bEnable := stAutomaticControlSettings.bEnableVelocityFeedForwardControl,
	fInput_ms := fbMotionReferenceGenerator.fVelocityReference_ms,
	fDisplacment_cc := stParam.fDisplacment_cc,
	stOpenLoopControlSettings := stOpenLoopControlSettings,
	rCircumference := 0.07 * 3.14,
	rTransmission := 1.0
);

fbResetIntegralController(
	stClosedLoopControlSettings := stClosedLoopControlSettings,
	fPositionError_m := fbClosedLoopPositionControl.xCylErrormm,
	fVelocityReference_ms := fbMotionReferenceGenerator.fVelocityReference_ms
);

rWinchPosRad := 3.141 * G_Sensors.fWinchEncoderPosition / 180; 
fbHeightCalc(
	xCyl := G_Sensors.fPositionCylPiston,
	winchAngleRad :=rWinchPosRad,
	hZero := G_HeightCorrection.rZeroOffset,
	wheelHeight := 0.330,
	totalDistance := 1.451,
	spoolRadius := 0.04575);
	
G_HeightCorrection.rActual := fbHeightCalc.height;

IF G_HeightCorrection.xCorrectHeight=TRUE THEN
	rSetPos := G_HeightCorrection.rDesiredHeight;
	rActPos := G_HeightCorrection.rActual;
ELSE
	rSetPos := fbMotionReferenceGenerator.fPositionReference_m;
	rActPos := G_HeightCorrection.rActual;
END_IF


fbClosedLoopPositionControl(
	EnablePFC := stAutomaticControlSettings.bEnableClosedLoopPositionControl,
	PosRefm := rSetPos,
	VRefms := fbMotionReferenceGenerator.fVelocityReference_ms,
	PosFbm := rActPos,
	propGain := stClosedLoopControlSettings.fProportionalGain,
	integralGain := stClosedLoopControlSettings.fIntegralGain,
	maxPosError := stClosedLoopControlSettings.fMaxPositionError,
	EnableIntegral := stAutomaticControlSettings.bEnableIntegralController,
	ssMethodType := BOOL_TO_SINT(bEnable AND bStartMotion)
);

fVelocityReference_ms := fbMotionReferenceGenerator.fVelocityReference_ms;
fPositionReference_m := fbMotionReferenceGenerator.fPositionReference_m;
fTime := fbClock.fTime;
fPositionError_mm := fbClosedLoopPositionControl.xCylErrormm/1E3;

IF bEnable THEN
	fControlOutputNormalized := LIMIT(-1.0, (fbVelocityFeedForwardControl.fNormalizedOutput + fbClosedLoopPositionControl.SetValue), 1.0);
ELSE
	fControlOutputNormalized := 0.0;
END_IF

END_FUNCTION_BLOCK

// ---- Machine Control/Function blocks/FB_Clock.TcPOU
FUNCTION_BLOCK FB_Clock
VAR_INPUT
	bEnable 	: BOOL;
	bStart 		: BOOL;
	bStop 		: BOOL;
	fCycleTime  : LREAL;
END_VAR
VAR_OUTPUT
	fTime : LREAL;
END_VAR
VAR
END_VAR

IF bStart AND NOT(bStop) AND bEnable THEN
	fTime := fTime + fCycleTime;
ELSE
	fTime := 0.0;
END_IF

END_FUNCTION_BLOCK

// ---- Machine Control/Function blocks/FB_MotionReferenceGenerator_limit.TcPOU
FUNCTION_BLOCK FB_MotionReferenceGenerator_limit
VAR_INPUT
	bEnable 							: BOOL;
	stMotionReferenceGeneratorSettings  : ST_MotionReferenceGeneratorSettings;
	fClock_s							: LREAL;
END_VAR
VAR_OUTPUT
	fPositionReference_m	: LREAL;
	fVelocityReference_ms	: LREAL;
	fTotalMotionTime_s		: LREAL;
	bErrorSignal			: BOOL;
END_VAR
VAR
	fStartPosition_m		: LREAL;
	fStartVelocity_m		: LREAL;
	fPositionSetpoint_ms	: LREAL;
	fVelocitySetpoint_m		: LREAL;
	fTimeBeforeStarting_s	: LREAL;
	fRampTime_s				: LREAL;
	fHoldPositionTime_s		: LREAL;
	Error					: DINT;
	slopeExt				: LREAL;
	slopeRetr				: LREAL;
	tHold					: LREAL;
	x1						: LREAL;
	x4						: LREAL;
	x1_tmp					: LREAL;
	x1_tmp_tmp				: LREAL;
	x4_tmp					: LREAL;
	x4_tmp_tmp				: LREAL;
	x4_tmp_tmp_0			: LREAL;
	x1_tmp_0				: LREAL;
END_VAR

IF NOT(bEnable) THEN
	RETURN;
END_IF

// LIMIT function: https://help.codesys.com/api-content/2/codesys/3.5.12.0/en/_cds_operator_limit/
fStartPosition_m := LIMIT(stMotionReferenceGeneratorSettings.fMinPosition, stMotionReferenceGeneratorSettings.fStartPosition_m, stMotionReferenceGeneratorSettings.fMaxPosition);
fStartVelocity_m := LIMIT(0.0, stMotionReferenceGeneratorSettings.fStartVelocity_m, stMotionReferenceGeneratorSettings.fMaxVelocity);
fPositionSetpoint_ms := LIMIT(stMotionReferenceGeneratorSettings.fMinPosition, stMotionReferenceGeneratorSettings.fPositionSetpoint_ms, stMotionReferenceGeneratorSettings.fMaxPosition);
fVelocitySetpoint_m := LIMIT(0.0, stMotionReferenceGeneratorSettings.fVelocitySetpoint_m, stMotionReferenceGeneratorSettings.fMaxVelocity);
fTimeBeforeStarting_s := LIMIT(0.0, stMotionReferenceGeneratorSettings.fTimeBeforeStarting_s, 10.0);
fRampTime_s := LIMIT(0.0, stMotionReferenceGeneratorSettings.fRampTime_s, 10.0);
fHoldPositionTime_s := LIMIT(0.0, stMotionReferenceGeneratorSettings.fHoldPositionTime_s, 60.0);

slopeExt := fStartVelocity_m - fVelocitySetpoint_m;

slopeRetr := ( -fVelocitySetpoint_m) - fStartVelocity_m;

tHold := ((fPositionSetpoint_ms - fStartPosition_m) - (((fVelocitySetpoint_m * fVelocitySetpoint_m) - (fStartVelocity_m * fStartVelocity_m)) / (fVelocitySetpoint_m / fRampTime_s))) / fVelocitySetpoint_m;

IF tHold < 0.0  THEN 
    bErrorSignal := TRUE;
ELSE 
    bErrorSignal := FALSE;
END_IF;

x1_tmp_tmp := fTimeBeforeStarting_s + fRampTime_s;
x1_tmp := x1_tmp_tmp - fTimeBeforeStarting_s;
x1_tmp_0 := slopeExt / fRampTime_s;
x1 := ((x1_tmp * fStartVelocity_m) + fStartPosition_m) - ((x1_tmp_0 * (x1_tmp * x1_tmp)) / 2.0);

x4_tmp_tmp := x1_tmp_tmp + tHold;
x4_tmp_tmp_0 := x4_tmp_tmp + fRampTime_s;
x4_tmp := x4_tmp_tmp_0 + fHoldPositionTime_s;
x1_tmp := x4_tmp + fRampTime_s;
x4 := x1_tmp - x4_tmp;
x4 := (fPositionSetpoint_ms - (x4 * fStartVelocity_m)) + (((slopeRetr / fRampTime_s) * (x4 * x4)) / 2.0);

IF Error = 1 THEN 
    fPositionReference_m := fStartPosition_m;
    fVelocityReference_ms := fStartVelocity_m;
ELSIF (fClock_s >= 0.0) AND (fClock_s < fTimeBeforeStarting_s) THEN 
    fPositionReference_m := fStartPosition_m;
    fVelocityReference_ms := fStartVelocity_m;
ELSIF (fClock_s >= fTimeBeforeStarting_s) AND (fClock_s < x1_tmp_tmp) THEN 
    slopeRetr := fClock_s - fTimeBeforeStarting_s;
    fPositionReference_m := ((slopeRetr * fStartVelocity_m) + fStartPosition_m) - ((x1_tmp_0 * (slopeRetr * slopeRetr)) / 2.0);
    fVelocityReference_ms := fStartVelocity_m - (x1_tmp_0 * slopeRetr);
ELSIF (fClock_s >= x1_tmp_tmp) AND (fClock_s < x4_tmp_tmp) THEN 
    fPositionReference_m := ((fClock_s - x1_tmp_tmp) * fVelocitySetpoint_m) + x1;
    fVelocityReference_ms := fVelocitySetpoint_m;
ELSIF (fClock_s >= x4_tmp_tmp) AND (fClock_s < x4_tmp_tmp_0) THEN 
    slopeRetr := fClock_s - x4_tmp_tmp;
    fPositionReference_m := ((((x4_tmp_tmp - x1_tmp_tmp) * fVelocitySetpoint_m) + x1) + (slopeRetr * fVelocitySetpoint_m)) + ((x1_tmp_0 * (slopeRetr * slopeRetr)) / 2.0);
    fVelocityReference_ms := (slopeRetr * (slopeExt / fRampTime_s)) + fVelocitySetpoint_m;
ELSIF (fClock_s >= x4_tmp_tmp_0) AND (fClock_s < x4_tmp) THEN 
    fPositionReference_m := fPositionSetpoint_ms;
    fVelocityReference_ms := fStartVelocity_m;
ELSIF (fClock_s >= x4_tmp) AND (fClock_s < x1_tmp) THEN 
    slopeExt := fClock_s - x4_tmp;
    slopeRetr := slopeRetr / fRampTime_s;
    fPositionReference_m := (fPositionSetpoint_ms - (slopeExt * fStartVelocity_m)) + ((slopeRetr * (slopeExt * slopeExt)) / 2.0);
    fVelocityReference_ms := (slopeExt * slopeRetr) + fStartVelocity_m;
ELSE 
    x1_tmp_0 := x1_tmp + tHold;

    IF (fClock_s >= x1_tmp) AND (fClock_s < x1_tmp_0) THEN 
        fPositionReference_m := x4 - ((fClock_s - x1_tmp) * fVelocitySetpoint_m);
        fVelocityReference_ms :=  -fVelocitySetpoint_m;
    ELSIF (fClock_s >= x1_tmp_0) AND (fClock_s < (((((((fTimeBeforeStarting_s + fRampTime_s) + tHold) + fRampTime_s) + fHoldPositionTime_s) + fRampTime_s) + tHold) + fRampTime_s)) THEN 
        slopeExt := fClock_s - x1_tmp_0;
        slopeRetr := slopeRetr / fRampTime_s;
        fPositionReference_m := ((x4 - ((x1_tmp_0 - x1_tmp) * fVelocitySetpoint_m)) - (slopeExt * fVelocitySetpoint_m)) - ((slopeRetr * (slopeExt * slopeExt)) / 2.0);
        fVelocityReference_ms := ( -fVelocitySetpoint_m) - (slopeExt * slopeRetr);
    ELSE 
        fPositionReference_m := fStartPosition_m;
        fVelocityReference_ms := fStartVelocity_m;
    END_IF;

END_IF;

fTotalMotionTime_s := ((((((fTimeBeforeStarting_s + fRampTime_s) + tHold) + fRampTime_s) + fHoldPositionTime_s) + fRampTime_s) + tHold) + fRampTime_s;

END_FUNCTION_BLOCK

// ---- Machine Control/Function blocks/FB_FeedforwardWinch.TcPOU
FUNCTION_BLOCK FB_FeedforwardWinch
VAR_INPUT
	bEnable		: BOOL;
	fInput_ms	: LREAL;
	fDisplacment_cc : LREAL;
	rCircumference : REAL;
	stOpenLoopControlSettings : ST_OpenLoopControlSettings;
	rTransmission : REAL;
END_VAR
VAR_OUTPUT
	fNormalizedOutput: LREAL;
END_VAR
VAR
	fFlowReference_lmin : LREAL;
	fRads : LREAL;
END_VAR

fRads := fInput_ms * 3.14 * 2 * rTransmission / (rCircumference);
fFlowReference_lmin := (fDisplacment_cc*1E-5*fRads/(2*3.14))*60000;

IF bEnable THEN 
    fNormalizedOutput := (fFlowReference_lmin) / stOpenLoopControlSettings.fMaxFlowCapacity;
ELSE 
    fNormalizedOutput := 0.0;
END_IF;

IF fNormalizedOutput > 1.0 THEN
    fNormalizedOutput := 1.0;
ELSIF fNormalizedOutput < -1.0 THEN 
    fNormalizedOutput := -1.0;
END_IF;

END_FUNCTION_BLOCK

// ---- Machine Control/Function blocks/FB_ResetIntegralController.TcPOU
FUNCTION_BLOCK FB_ResetIntegralController
VAR_INPUT
	stClosedLoopControlSettings : ST_ClosedLoopControlSettings;
	fVelocityReference_ms	: LREAL;
	fPositionError_m		: LREAL;
END_VAR
VAR_OUTPUT
	bReset: BOOL;
END_VAR
VAR
END_VAR

IF ABS(fVelocityReference_ms) > 0.0 THEN 
    bReset := FALSE;
ELSIF ABS(fPositionError_m) > stClosedLoopControlSettings.fMaxPositionError THEN 
    bReset := FALSE;
ELSE 
    bReset := TRUE;
END_IF;

END_FUNCTION_BLOCK

// ---- Machine Control/Function blocks/FB_CylController.TcPOU
FUNCTION_BLOCK FB_CylController
VAR_INPUT
	ssMethodType: SINT;
	EnablePFC: BOOL;
	PosRefm: LREAL;
	PosFbm: LREAL;
	propGain: LREAL;
	vRefms: LREAL;
	integralGain: LREAL;
	EnableIntegral: BOOL;
	maxPosError: LREAL;
END_VAR
VAR_OUTPUT
	xCylErrormm: LREAL;
	SetValue: LREAL;
END_VAR
VAR
	rtb_Reset: LREAL;
	rtb_u_FB: LREAL;
	rtb_Saturation1: LREAL;
	c_DiscreteTimeIntegrator_DS: LREAL;
	Delay_DSTATE: ARRAY[0..1] OF LREAL;
END_VAR



CASE ssMethodType OF
    SS_INITIALIZE: 
        (* SystemInitialize for Atomic SubSystem: '<Root>/CylController' *)
        (* InitializeConditions for Delay: '<S1>/Delay' *)
        Delay_DSTATE[0] := 0.0;
        Delay_DSTATE[1] := 0.0;
        (* SystemInitialize for Atomic SubSystem: '<S1>/FB_ClosedLoopControl' *)
        (* InitializeConditions for DiscreteIntegrator: '<S2>/Discrete-Time Integrator' *)
        c_DiscreteTimeIntegrator_DS := 0.0;
        (* End of SystemInitialize for SubSystem: '<S1>/FB_ClosedLoopControl' *)
        (* End of SystemInitialize for SubSystem: '<Root>/CylController' *)
		SetValue := 0.0;
		c_DiscreteTimeIntegrator_DS := 0.0;
		PosRefm := 0.0;
		vRefms := 0.0;
    SS_STEP: 
        (* Outputs for Atomic SubSystem: '<Root>/CylController' *)
        (* Outputs for Atomic SubSystem: '<S1>/FB_ResetIntegralController' *)
        (* MATLAB Function: '<S3>/ResetIntegralController' *)
        (* MATLAB Function 'CylController/FB_ResetIntegralController/ResetIntegralController': '<S4>:1' *)
        (* '<S4>:1:3' if abs(vRef) > 0 || abs(exCyl) > exCylMax *)

        IF ABS(vRefms) > 0.0 THEN 
            ;
            ;
        ELSIF ABS(Delay_DSTATE[0]) > (0.001 * maxPosError) THEN 
            ;
            ;
        ELSE 
            (* Outputs for Atomic SubSystem: '<S1>/FB_ClosedLoopControl' *)
            (* DiscreteIntegrator: '<S2>/Discrete-Time Integrator' *)
            (* '<S4>:1:5' else *)
            (* '<S4>:1:6' Reset = 1; *)
            c_DiscreteTimeIntegrator_DS := 0.0;
            (* End of Outputs for SubSystem: '<S1>/FB_ClosedLoopControl' *)
        END_IF;

        (* End of MATLAB Function: '<S3>/ResetIntegralController' *)
        (* End of Outputs for SubSystem: '<S1>/FB_ResetIntegralController' *)
        

        (* Outputs for Atomic SubSystem: '<S1>/FB_ClosedLoopControl' *)
        (* DiscreteIntegrator: '<S2>/Discrete-Time Integrator' *)

        IF c_DiscreteTimeIntegrator_DS >= 1.0 THEN 
            c_DiscreteTimeIntegrator_DS := 1.0;
        ELSIF c_DiscreteTimeIntegrator_DS <= -1.0 THEN 
            c_DiscreteTimeIntegrator_DS := -1.0;
        END_IF;

        (* Sum: '<S2>/Sum1' *)
        rtb_Reset := PosRefm - PosFbm;
        (* Switch: '<S2>/Switch' incorporates:
         *  Constant: '<S2>/Constant'
         *  DiscreteIntegrator: '<S2>/Discrete-Time Integrator' *)

        IF EnableIntegral THEN 
            rtb_u_FB := c_DiscreteTimeIntegrator_DS;
        ELSE 
            rtb_u_FB := 0.0;
        END_IF;

        (* End of Switch: '<S2>/Switch' *)
        

        (* Sum: '<S2>/Sum5' incorporates:
         *  Product: '<S2>/Product' *)
        rtb_u_FB := (propGain * rtb_Reset) + rtb_u_FB;
        (* Saturate: '<S2>/Saturation1' *)

        IF rtb_u_FB > 1.0 THEN 
            rtb_Saturation1 := 1.0;
        ELSIF rtb_u_FB >= -1.0 THEN 
            rtb_Saturation1 := rtb_u_FB;
        ELSE 
            rtb_Saturation1 := -1.0;
        END_IF;

        (* End of Saturate: '<S2>/Saturation1' *)
        

        (* Switch: '<S2>/Switch1' *)

        IF EnablePFC THEN 
            (* Outport: '<Root>/Set Value' *)
            SetValue := rtb_Saturation1;
        ELSE 
            (* Outport: '<Root>/Set Value' incorporates:
             *  Constant: '<S2>/Constant1' *)
            SetValue := 0.0;
        END_IF;

        (* End of Switch: '<S2>/Switch1' *)
        

        (* Update for DiscreteIntegrator: '<S2>/Discrete-Time Integrator' incorporates:
         *  Product: '<S2>/Divide'
         *  Product: '<S2>/Product2'
         *  Sum: '<S2>/Sum2'
         *  Sum: '<S2>/Sum3' *)
        c_DiscreteTimeIntegrator_DS := (((((rtb_Saturation1 - rtb_u_FB) / propGain) + rtb_Reset) * integralGain) * 0.001) + c_DiscreteTimeIntegrator_DS;

        IF c_DiscreteTimeIntegrator_DS >= 1.0 THEN 
            c_DiscreteTimeIntegrator_DS := 1.0;
        ELSIF c_DiscreteTimeIntegrator_DS <= -1.0 THEN 
            c_DiscreteTimeIntegrator_DS := -1.0;
        END_IF;

        (* End of Update for DiscreteIntegrator: '<S2>/Discrete-Time Integrator' *)
        (* End of Outputs for SubSystem: '<S1>/FB_ClosedLoopControl' *)
        

        (* Update for Delay: '<S1>/Delay' *)
        Delay_DSTATE[0] := Delay_DSTATE[1];
        Delay_DSTATE[1] := rtb_Reset;
        (* Outport: '<Root>/xCylError [mm]' incorporates:
         *  Gain: '<S1>/Gain' *)
        xCylErrormm := 1000.0 * rtb_Reset;
        (* End of Outputs for SubSystem: '<Root>/CylController' *)
END_CASE;

END_FUNCTION_BLOCK

// ---- Machine Control/Function blocks/FB_AutomaticControl.TcPOU
FUNCTION_BLOCK FB_AutomaticControl
VAR_INPUT
	bEnable 							: BOOL;
	bStartMotion 						: BOOL;
	bStopMotion 						: BOOL;
	stMotionReferenceGeneratorSettings  : ST_MotionReferenceGeneratorSettings;
	stAutomaticControlSettings 			: ST_AutomaticControlSettings;
	stClosedLoopControlSettings 		: ST_ClosedLoopControlSettings;
	stOpenLoopControlSettings			: ST_OpenLoopControlSettings;
	stParam 							: ST_Parameters; 
	fPositionFeedback					: LREAL;
END_VAR
VAR_OUTPUT
	fTime : LREAL;
	fVelocityReference_ms : LREAL;
	fPositionReference_m : LREAL;
	fControlOutputNormalized : LREAL;
	fPositionError_mm : LREAL;
END_VAR
VAR
	fbClock : FB_Clock;	
	fbMotionReferenceGenerator 		: FB_MotionReferenceGenerator_limit;	
	fbVelocityFeedForwardControl 	: FB_FeedForwardCyl;
	fbResetIntegralController 		: FB_ResetIntegralController; 
	fbClosedLoopPositionControl 	: FB_CylController;
END_VAR

fbClock(
	bEnable := bEnable,
	bStart := bStartMotion,
	bStop := bStopMotion,
	fCycleTime := G_Parameters.stParam.fCyclicTime
);

fbMotionReferenceGenerator(
	bEnable := bEnable,
	stMotionReferenceGeneratorSettings := stMotionReferenceGeneratorSettings,
	fClock_s := fbClock.fTime
);

fbVelocityFeedForwardControl(
	Enable := stAutomaticControlSettings.bEnableVelocityFeedForwardControl,
	vRef_ms := fbMotionReferenceGenerator.fVelocityReference_ms,
	maxFlow_lmin := stOpenLoopControlSettings.fMaxFlowCapacity,
	cylOpeningForward := 0.00331,
	cylOpeningBackward := 0.00236,
);

(* fbResetIntegralController(
	stClosedLoopControlSettings := stClosedLoopControlSettings,
	fPositionError_m := fbClosedLoopPositionControl.fPositionError,
	fVelocityReference_ms := fbMotionReferenceGenerator.fVelocityReference_ms
);*)

(*fbClosedLoopPositionControl(
	bEnable := stAutomaticControlSettings.bEnableClosedLoopPositionControl,
	stParam := stParam,
	stClosedLoopControlSettings := stClosedLoopControlSettings,		
	bActivateIntegralController := stAutomaticControlSettings.bEnableIntegralController,
	bIntegralControllReset := fbResetIntegralController.bReset,
	fInput_m := fbMotionReferenceGenerator.fPositionReference_m,
	fFeedback_m := fPositionFeedback
);*)


fVelocityReference_ms := fbMotionReferenceGenerator.fVelocityReference_ms;
fPositionReference_m := fbMotionReferenceGenerator.fPositionReference_m;
fTime := fbClock.fTime;


fbClosedLoopPositionControl(
	EnablePFC := stAutomaticControlSettings.bEnableClosedLoopPositionControl,
	PosRefm := fbMotionReferenceGenerator.fPositionReference_m,
	VRefms := fbMotionReferenceGenerator.fVelocityReference_ms,
	PosFbm := fPositionFeedback,
	propGain := stClosedLoopControlSettings.fProportionalGain,
	integralGain := stClosedLoopControlSettings.fIntegralGain,
	maxPosError := stClosedLoopControlSettings.fMaxPositionError,
	EnableIntegral := stAutomaticControlSettings.bEnableIntegralController,
	ssMethodType := BOOL_TO_SINT(bEnable AND bStartMotion)
);

fPositionError_mm := fbClosedLoopPositionControl.xCylerrormm;

IF bEnable THEN
	fControlOutputNormalized := LIMIT(-1.0, (fbVelocityFeedForwardControl.FeedfowardOutput + fbClosedLoopPositionControl.SetValue), 1.0);
ELSE
	fControlOutputNormalized := 0.0;
END_IF

END_FUNCTION_BLOCK

// ---- Machine Control/Function blocks/FB_FeedForwardCyl.TcPOU
FUNCTION_BLOCK FB_FeedForwardCyl
VAR_INPUT
	Enable: BOOL;
	vRef_ms: LREAL;
	maxFlow_lmin: LREAL;
	cylOpeningForward: LREAL;
	cylOpeningBackward: LREAL;
END_VAR
VAR_OUTPUT
	FeedfowardOutput: LREAL;
END_VAR
VAR
	rtb_Switch: LREAL;
END_VAR


(* Outputs for Atomic SubSystem: '<Root>/FeedForward' *)
(* Switch: '<S1>/Switch1' *)

IF Enable THEN 
    (* Switch: '<S1>/Switch' incorporates:
     *  Constant: '<S1>/Constant'
     *  Product: '<S1>/Product1'
     *  Product: '<S1>/Product2'
     *  RelationalOperator: '<S1>/Relational Operator' *)

    IF vRef_ms >= 0.0 THEN 
        rtb_Switch := cylOpeningForward * vRef_ms;
    ELSE 
        rtb_Switch := vRef_ms * cylOpeningBackward;
    END_IF;

    (* End of Switch: '<S1>/Switch' *)
    

    (* Outport: '<Root>/FeedfowardOutput' incorporates:
     *  Constant: '<S1>/Constant2'
     *  Product: '<S1>/Divide'
     *  Product: '<S1>/Product' *)
    FeedfowardOutput := (60000.0 * rtb_Switch) / maxFlow_lmin;
ELSE 
    (* Outport: '<Root>/FeedfowardOutput' incorporates:
     *  Constant: '<S1>/Constant1' *)
    FeedfowardOutput := 0.0;
END_IF;

(* End of Switch: '<S1>/Switch1' *)
(* End of Outputs for SubSystem: '<Root>/FeedForward' *)

END_FUNCTION_BLOCK

// ---- HMI/Function blocks/FB_ModifyAutomaticControlSettings.TcPOU
FUNCTION_BLOCK FB_ModifyAutomaticControlSettings
VAR_INPUT
	stParamOpenLoopControllSettings 	: REFERENCE TO ST_OpenLoopControlSettings;
	stParamClosedLoopControllSettings 	: REFERENCE TO ST_ClosedLoopControlSettings;
	stModify 							: ST_ModifyAutomaticControlSettings;
END_VAR
VAR_OUTPUT
END_VAR
VAR
END_VAR

IF stModify.bSetNewMaxFlowCapacity THEN
	stParamOpenLoopControllSettings.fMaxFlowCapacity := stModify.fNewMaxFlowCapacity;
	stModify.bSetNewMaxFlowCapacity := FALSE;
END_IF

IF stModify.bSetNewProportionalGain THEN
	stParamClosedLoopControllSettings.fProportionalGain := stModify.fNewProportionalGain;
	stModify.bSetNewProportionalGain := FALSE;
END_IF

IF stModify.bSetNewIntegralGain THEN
	stParamClosedLoopControllSettings.fIntegralGain := stModify.fNewIntegralGain;
	stModify.bSetNewIntegralGain := FALSE;
END_IF

IF stModify.bSetNewMaxPositionError THEN
	stParamClosedLoopControllSettings.fMaxPositionError:= stModify.fNewMaxPositionError;
	stModify.bSetNewMaxPositionError := FALSE;
END_IF

END_FUNCTION_BLOCK

// ---- Outputs/P_Outputs.TcPOU
PROGRAM P_Outputs
VAR
	fbWinchValveOutput 		: FB_ValveOutput;
	fbCylValveOutput 		: FB_ValveOutput;
END_VAR

///////////////////// Winch //////////////////////////////
G_Outputs.stWinchValveOutput.bEnable := G_Work.bManualMode OR G_Work.bAutoMode; 

fbWinchValveOutput(
	bEnable := (G_Work.bWinchEnable OR G_Work.fWinchTime > 0.0) AND G_Hmi.bWinchEnable,
	bDeadBandCompOn := G_Parameters.stParam.bDeadBandCompOn,
	stValveDeadBand := G_Parameters.stParam.stWinchValveDeadBand,
	fNormalizedInput := G_Work.fWinchControlInput,
	nOutput => G_Outputs.stWinchValveOutput.nValveOutput
);

///////////////////// Cylinder //////////////////////////////
G_Outputs.stCylValveOutput.bEnable := G_Work.bManualMode OR G_Work.bAutoMode;

fbCylValveOutput(
	bEnable := (G_Work.bCylEnable OR G_Work.fCylTime > 0.0) AND G_Hmi.bCylEnable,
	bDeadBandCompOn := G_Parameters.stParam.bDeadBandCompOn,
	stValveDeadBand := G_Parameters.stParam.stCylValveDeadBand,
	fNormalizedInput := G_Work.fCylControlInput,
	nOutput => G_Outputs.stCylValveOutput.nValveOutput
);

END_PROGRAM

// ---- Outputs/Function blocks/FB_ValveOutput.TcPOU
FUNCTION_BLOCK FB_ValveOutput
VAR_INPUT
	bEnable 			: BOOL;
	bDeadBandCompOn 	: BOOL;
	stValveDeadBand 	: ST_ValveDeadBand;
	fNormalizedInput 	: LREAL;
END_VAR
VAR_OUTPUT
	bEnableValveOutput : BOOL;
	nOutput : INT; 
END_VAR
VAR
	nOffset 	: INT := 19660;
	nMaxValue	: INT := 29490;
	nMinValue 	: INT :=  9830;
	nTempOutput : INT;
END_VAR

IF	bDeadBandCompOn THEN
	IF fNormalizedInput > 0.0 THEN
		nTempOutput := LREAL_TO_INT(ABS(fNormalizedInput*(stValveDeadBand.fPosMax - stValveDeadBand.fPosMin) + stValveDeadBand.fPosMin));
	ELSIF fNormalizedInput < 0.0 THEN
		nTempOutput := LREAL_TO_INT(ABS(fNormalizedInput*(stValveDeadBand.fNegMax - stValveDeadBand.fNegMin) - stValveDeadBand.fNegMin));
	ELSE
		nTempOutput := nOffset;
	END_IF
ELSE
	IF fNormalizedInput > 0.0 THEN
		nTempOutput := LREAL_TO_INT(ABS(fNormalizedInput*(32767.0 - 19660.0) + 19660.0));
	ELSIF fNormalizedInput < 0.0 THEN
		nTempOutput := LREAL_TO_INT(ABS(fNormalizedInput*(0 - 19660.0) - 19660.0));
	ELSE
		nTempOutput := nOffset;
	END_IF	
END_IF	

IF bEnable THEN
	nOutput := LIMIT(nMinValue, nTempOutput, nMaxValue);
	bEnableValveOutput := TRUE; 
ELSE 	
	nOutput := nOffset;
	bEnableValveOutput := FALSE;	
END_IF

END_FUNCTION_BLOCK

// ---- Inputs/Functions/F_DegToRad.TcPOU
FUNCTION F_DegToRad : LREAL
VAR_INPUT
	fInputDeg 	: LREAL;
END_VAR
VAR
	fPi 		:LREAL := 3.14159265359;
END_VAR

F_DegToRad := fInputDeg*(fPi/180);

END_FUNCTION

// ---- Machine Control/Function blocks/FB_ClosedLoopControl.TcPOU
FUNCTION_BLOCK FB_ClosedLoopControl
VAR_INPUT
	bEnable						: BOOL;
	stParam 					: ST_Parameters; 
	stClosedLoopControlSettings : ST_ClosedLoopControlSettings;
	bActivateIntegralController	: BOOL;
	bIntegralControllReset		: BOOL;
	fInput_m					: LREAL;
	fFeedback_m					: LREAL;
END_VAR
VAR_OUTPUT
	fNormalizedOutput	: LREAL;
	fPositionError		: LREAL;
END_VAR
VAR
	rtb_u_FB					: LREAL;
	rtb_Saturation1				: LREAL;
	c_DiscreteTimeIntegrator_DS	: LREAL;
END_VAR

fPositionError := fInput_m - fFeedback_m;

IF bIntegralControllReset THEN 
	c_DiscreteTimeIntegrator_DS := 0.0;
END_IF;

IF c_DiscreteTimeIntegrator_DS >= 1.0 THEN 
	c_DiscreteTimeIntegrator_DS := 1.0;
ELSIF c_DiscreteTimeIntegrator_DS <= -1.0 THEN 
	c_DiscreteTimeIntegrator_DS := -1.0;
END_IF;

IF bActivateIntegralController THEN 
	rtb_u_FB := c_DiscreteTimeIntegrator_DS;
ELSE 
	rtb_u_FB := 0.0;
END_IF;

rtb_u_FB := (stClosedLoopControlSettings.fProportionalGain * fPositionError) + rtb_u_FB;

IF rtb_u_FB > 1.0 THEN 
	rtb_Saturation1 := 1.0;
ELSIF rtb_u_FB >= -1.0 THEN 
	rtb_Saturation1 := rtb_u_FB;
ELSE 
	rtb_Saturation1 := -1.0;
END_IF;

IF bEnable THEN 
	fNormalizedOutput := rtb_Saturation1;
ELSE 
	fNormalizedOutput := 0.0;
END_IF;

c_DiscreteTimeIntegrator_DS := (((((rtb_Saturation1 - rtb_u_FB) / stClosedLoopControlSettings.fProportionalGain) + fPositionError) * stClosedLoopControlSettings.fIntegralGain) * stParam.fCyclicTime) + c_DiscreteTimeIntegrator_DS;

IF c_DiscreteTimeIntegrator_DS >= 1.0 THEN 
	c_DiscreteTimeIntegrator_DS := 1.0;
ELSIF c_DiscreteTimeIntegrator_DS <= -1.0 THEN 
	c_DiscreteTimeIntegrator_DS := -1.0;
END_IF;

END_FUNCTION_BLOCK

// ---- Machine Control/Function blocks/FB_OpenLoopControl.TcPOU
FUNCTION_BLOCK FB_OpenLoopControl
VAR_INPUT
	bEnable		: BOOL;
	fInput_ms	: LREAL;
	stOpenLoopControlSettings : ST_OpenLoopControlSettings;
END_VAR
VAR_OUTPUT
	fNormalizedOutput: LREAL;
END_VAR
VAR
	fFlowReference_m3s : LREAL;
	fM3sToLmin : LREAL := 60000;
END_VAR

IF fInput_ms >= 0.0 THEN 
    fFlowReference_m3s := stOpenLoopControlSettings.fBoreArea * fInput_ms;
ELSE 
    fFlowReference_m3s := fInput_ms * stOpenLoopControlSettings.fAnnulusArea;
END_IF;

IF bEnable THEN 
    fNormalizedOutput := (fM3sToLmin * fFlowReference_m3s) / stOpenLoopControlSettings.fMaxFlowCapacity;
ELSE 
    fNormalizedOutput := 0.0;
END_IF;

IF fNormalizedOutput > 1.0 THEN 
    fNormalizedOutput := 1.0;
ELSIF fNormalizedOutput < -1.0 THEN 
    fNormalizedOutput := -1.0;
END_IF;

END_FUNCTION_BLOCK

// ---- Machine Control/Function blocks/FB_OpenLoopControlWinch.TcPOU
FUNCTION_BLOCK FB_OpenLoopControlWinch
VAR_INPUT
	bEnable		: BOOL;
	fInput_ms	: LREAL;
	fDisplacment_cc : LREAL;
	fLin_m_ToRot_deg_Scaling : LREAL;
	stOpenLoopControlSettings : ST_OpenLoopControlSettings;
END_VAR
VAR_OUTPUT
	fNormalizedOutput: LREAL;
END_VAR
VAR
	fFlowReference_lmin : LREAL;
	fRads : LREAL;
END_VAR

fRads := (fInput_ms/fLin_m_ToRot_deg_Scaling)*3.14/180;
//fFlowReference_lmin := (fDisplacment_cc*(fRads/(2*3.14)*60))/1000;
fFlowReference_lmin := (fDisplacment_cc*1E-5*fRads/(2*3.14))*60000;

IF bEnable THEN 
    fNormalizedOutput := (fFlowReference_lmin) / stOpenLoopControlSettings.fMaxFlowCapacity;
ELSE 
    fNormalizedOutput := 0.0;
END_IF;

IF fNormalizedOutput > 1.0 THEN 
    fNormalizedOutput := 1.0;
ELSIF fNormalizedOutput < -1.0 THEN 
    fNormalizedOutput := -1.0;
END_IF;

END_FUNCTION_BLOCK

// ---- Machine Control/Function blocks/FB_ValveOutputGenerator.TcPOU
FUNCTION_BLOCK FB_ValveOutputGenerator
VAR_INPUT
	bEnable: BOOL;
	stValveOutputGeneratorSettings : ST_ValveOutputGeneratorSettings;
	fClock_s: LREAL;
END_VAR
VAR_OUTPUT
	fNormalizedValveOutputRef: LREAL;
	fTotalMotionTime_s: LREAL;
END_VAR
VAR
	fInitialValveOpening: LREAL;
	fValveOpeningSetPoint: LREAL;
	fTimeBeforeStarting_s: LREAL;
	fRampTime_s: LREAL;
	fHoldTime_s: LREAL;
	fWaitTime_s: LREAL;
	slopeExt: LREAL;
	slopeRetr: LREAL;
	Error: DINT;
	tmp: LREAL;
	temp1: LREAL;
END_VAR

fInitialValveOpening	:= stValveOutputGeneratorSettings.fInitialValveOpening;
fValveOpeningSetPoint	:= stValveOutputGeneratorSettings.fValveOpeningSetPoint;
fTimeBeforeStarting_s	:= stValveOutputGeneratorSettings.fTimeBeforeStarting_s;
fRampTime_s				:= stValveOutputGeneratorSettings.fRampTime_s;
fHoldTime_s				:= stValveOutputGeneratorSettings.fHoldTime_s;
fWaitTime_s				:= stValveOutputGeneratorSettings.fWaitTime_s;

(* Outputs for Atomic SubSystem: '<Root>/FB_AutomaticValveOutputGenerator' *)
(* Saturate: '<S1>/Saturation2' *)

IF fValveOpeningSetPoint > 1.0 THEN 
    fNormalizedValveOutputRef := 1.0;
ELSIF fValveOpeningSetPoint >= 0.0 THEN 
    fNormalizedValveOutputRef := fValveOpeningSetPoint;
ELSE 
    fNormalizedValveOutputRef := 0.0;
END_IF;

(* End of Saturate: '<S1>/Saturation2' *)


(* MATLAB Function: '<S1>/AutomaticValveOutputGenerator' *)
(* MATLAB Function 'FB_AutomaticValveOutputGenerator/AutomaticValveOutputGenerator': '<S2>:1' *)
(* '<S2>:1:2' us=u_ref; *)
(* '<S2>:1:3' slopeExt=u0-us; *)
slopeExt := fInitialValveOpening - fNormalizedValveOutputRef;
(* '<S2>:1:4' slopeRetr=-us-u0; *)
slopeRetr := ( -fNormalizedValveOutputRef) - fInitialValveOpening;
(* '<S2>:1:6' if tHold < 0 *)

IF fHoldTime_s < 0.0 THEN 
    (* '<S2>:1:7' Error = 1; *)
    Error := 1;
ELSE 
    (* '<S2>:1:8' else *)
    (* '<S2>:1:9' Error = 0; *)
    Error := 0;
END_IF;

(* '<S2>:1:12' t1=tRamp; *)
(* '<S2>:1:13' t2=tHold; *)
(* '<S2>:1:14' t3=tRamp; *)
(* '<S2>:1:15' t4=tWait; *)
(* '<S2>:1:16' t5=t1; *)
(* '<S2>:1:17' t6=t2; *)
(* '<S2>:1:18' t7=t3; *)
(* '<S2>:1:20' if Error == 1 *)

IF Error = 1 THEN 
    (* '<S2>:1:21' u = u0; *)
    fNormalizedValveOutputRef := fInitialValveOpening;
ELSIF (fClock_s >= 0.0) AND (fClock_s < fTimeBeforeStarting_s) THEN 
    (* '<S2>:1:22' elseif t>=0 && t<t0 *)
    (* '<S2>:1:23' u = u0; *)
    fNormalizedValveOutputRef := fInitialValveOpening;
ELSE 
    tmp := fTimeBeforeStarting_s + fRampTime_s;

    IF (fClock_s >= fTimeBeforeStarting_s) AND (fClock_s < tmp) THEN 
        (* '<S2>:1:24' elseif t>=t0 && t<(t0+t1) *)
        (* '<S2>:1:25' u = u0-(slopeExt/t1)*(t-t0); *)
        fNormalizedValveOutputRef := fInitialValveOpening - ((slopeExt / fRampTime_s) * (fClock_s - fTimeBeforeStarting_s));
    ELSE 
        temp1 := tmp + fHoldTime_s;

        IF (fClock_s < tmp) OR (fClock_s >= temp1) THEN 
            tmp := temp1 + fRampTime_s;

            IF (fClock_s >= temp1) AND (fClock_s < tmp) THEN 
                (* '<S2>:1:28' elseif t>=(t0+t1+t2) && t<(t0+t1+t2+t3) *)
                (* '<S2>:1:29' u = us+(slopeExt/t3)*(t-(t0+t1+t2)); *)
                fNormalizedValveOutputRef := ((fClock_s - temp1) * (slopeExt / fRampTime_s)) + fNormalizedValveOutputRef;
            ELSE 
                temp1 := tmp + fWaitTime_s;

                IF (fClock_s >= tmp) AND (fClock_s < temp1) THEN 
                    (* '<S2>:1:30' elseif t>=(t0+t1+t2+t3) && t<(t0+t1+t2+t3+t4) *)
                    (* '<S2>:1:31' u = u0; *)
                    fNormalizedValveOutputRef := fInitialValveOpening;
                ELSE 
                    tmp := temp1 + fRampTime_s;

                    IF (fClock_s >= temp1) AND (fClock_s < tmp) THEN 
                        (* '<S2>:1:32' elseif t>=(t0+t1+t2+t3+t4) && t<(t0+t1+t2+t3+t4+t5) *)
                        (* '<S2>:1:33' u = u0+(slopeRetr/t5)*(t-(t0+t1+t2+t3+t4)); *)
                        fNormalizedValveOutputRef := ((fClock_s - temp1) * (slopeRetr / fRampTime_s)) + fInitialValveOpening;
                    ELSE 
                        temp1 := tmp + fHoldTime_s;

                        IF (fClock_s >= tmp) AND (fClock_s < temp1) THEN 
                            (* '<S2>:1:34' elseif t>=(t0+t1+t2+t3+t4+t5) && t<(t0+t1+t2+t3+t4+t5+t6) *)
                            (* '<S2>:1:35' u = -us; *)
                            fNormalizedValveOutputRef :=  -fNormalizedValveOutputRef;
                        ELSIF (fClock_s >= temp1) AND (fClock_s < (temp1 + fRampTime_s)) THEN 
                            (* '<S2>:1:36' elseif t>=(t0+t1+t2+t3+t4+t5+t6) && t<(t0+t1+t2+t3+t4+t5+t6+t7) *)
                            (* '<S2>:1:37' u = -us-(slopeRetr/t3)*(t-(t0+t1+t2+t3+t4+t5+t6)); *)
                            fNormalizedValveOutputRef := ( -fNormalizedValveOutputRef) - ((fClock_s - temp1) * (slopeRetr / fRampTime_s));
                        ELSE 
                            (* '<S2>:1:38' else *)
                            (* '<S2>:1:39' u = u0; *)
                            fNormalizedValveOutputRef := fInitialValveOpening;
                        END_IF;

                    END_IF;

                END_IF;

            END_IF;

        END_IF;

    END_IF;

END_IF;

(* Switch: '<S1>/Switch' *)
(* '<S2>:1:42' T = t0+t1+t2+t3+t4+t5+t6+t7; *)

IF  NOT bEnable THEN 
    fNormalizedValveOutputRef := fInitialValveOpening;
END_IF;

(* End of Switch: '<S1>/Switch' *)


(* Saturate: '<S1>/Saturation' *)

IF fNormalizedValveOutputRef > 1.0 THEN 
    (* Outport: '<Root>/fNormalizedValveOutputRef' *)
    fNormalizedValveOutputRef := 1.0;
ELSIF fNormalizedValveOutputRef < -1.0 THEN 
    (* Outport: '<Root>/fNormalizedValveOutputRef' *)
    fNormalizedValveOutputRef := -1.0;
END_IF;

(* End of Saturate: '<S1>/Saturation' *)


(* Outport: '<Root>/fTotalMotionTime_s' incorporates:
 *  MATLAB Function: '<S1>/AutomaticValveOutputGenerator' *)
fTotalMotionTime_s := ((((((fTimeBeforeStarting_s + fRampTime_s) + fHoldTime_s) + fRampTime_s) + fWaitTime_s) + fRampTime_s) + fHoldTime_s) + fRampTime_s;
(* End of Outputs for SubSystem: '<Root>/FB_AutomaticValveOutputGenerator' *)

END_FUNCTION_BLOCK

// ---- Machine Control/Function blocks/FB_AutomaticControl_old.TcPOU
FUNCTION_BLOCK FB_AutomaticControl_old
VAR_INPUT
	bEnable								: BOOL;
	bStartMotion 						: BOOL;
	bStopMotion 						: BOOL;
	stValveOutputGeneratorSettings  	: ST_ValveOutputGeneratorSettings;
	stParam 		: ST_Parameters; 
END_VAR
VAR_OUTPUT
	fTime : LREAL;
	fNormalizedValveOpeningRefSignal : LREAL;
END_VAR
VAR
	fbClock 					: FB_Clock;	
	fbValveOutputGenerator 		: FB_ValveOutputGenerator;	
END_VAR

fbClock(
	bEnable := bEnable,
	bStart := bStartMotion,
	bStop := bStopMotion,
	fCycleTime := stParam.fCyclicTime
);

fbValveOutputGenerator(
	bEnable := bEnable,
	stValveOutputGeneratorSettings := stValveOutputGeneratorSettings,
	fClock_s := fbClock.fTime
);

fNormalizedValveOpeningRefSignal := fbValveOutputGenerator.fNormalizedValveOutputRef;
fTime := fbClock.fTime;

END_FUNCTION_BLOCK

// ---- Machine Control/Function blocks/FB_RampGen.TcPOU
FUNCTION_BLOCK FB_RampGen
VAR_INPUT
	ssMethodType: SINT;
	Enable: BOOL;
	x0m: LREAL;
	v0ms: LREAL;
	Position_SPm: LREAL;
	Velocity_SPms: LREAL;
	t0s: LREAL;
	tRamps: LREAL;
	tHoldPoss: LREAL;
	StartAuto: BOOL;
	StopAuto: BOOL;
END_VAR
VAR_OUTPUT
	PosRef: LREAL;
	VelRef: LREAL;
END_VAR
VAR
	Error: DINT;
	tHold: LREAL;
	x1: LREAL;
	x4: LREAL;
	rtb_Time: LREAL;
	rtb_Saturation3: LREAL;
	a_tmp: LREAL;
	a_tmp_tmp: LREAL;
	a_tmp_0: LREAL;
	a_tmp_tmp_0: LREAL;
	a_tmp_tmp_1: LREAL;
	a_tmp_tmp_2: LREAL;
	x1_tmp: LREAL;
	x4_tmp: LREAL;
	c_DiscreteTimeIntegrator_DS: LREAL;
END_VAR



CASE ssMethodType OF
    SS_INITIALIZE: 
        (* SystemInitialize for Atomic SubSystem: '<Root>/Subsystem' *)
        (* InitializeConditions for DiscreteIntegrator: '<S2>/Discrete-Time Integrator' *)
        c_DiscreteTimeIntegrator_DS := 0.0;
        (* End of SystemInitialize for SubSystem: '<Root>/Subsystem' *)
    SS_STEP: 
        (* Outputs for Atomic SubSystem: '<Root>/Subsystem' *)
        (* MATLAB Function: '<S2>/MATLAB Function' incorporates:
         *  DiscreteIntegrator: '<S2>/Discrete-Time Integrator' *)
        (* MATLAB Function 'Subsystem/MotionReferenceTime/MATLAB Function': '<S4>:1' *)
        (* '<S4>:1:3' if StartClock == 1 && ~StopClock *)

        IF StartAuto AND ( NOT StopAuto) THEN 
            (* '<S4>:1:4' Time = Clock; *)
            rtb_Time := c_DiscreteTimeIntegrator_DS;
        ELSE 
            (* '<S4>:1:5' else *)
            (* '<S4>:1:6' Time = 0.0; *)
            rtb_Time := 0.0;
        END_IF;

        (* End of MATLAB Function: '<S2>/MATLAB Function' *)
        

        (* Outputs for Atomic SubSystem: '<S1>/RampMotionProfileGenerator' *)
        (* Saturate: '<S3>/Saturation3' *)

        IF Position_SPm > 0.5 THEN 
            rtb_Saturation3 := 0.5;
        ELSIF Position_SPm >= 0.0 THEN 
            rtb_Saturation3 := Position_SPm;
        ELSE 
            rtb_Saturation3 := 0.0;
        END_IF;

        (* End of Saturate: '<S3>/Saturation3' *)
        

        (* Saturate: '<S3>/Saturation2' *)

        IF Velocity_SPms > 0.12 THEN 
            PosRef := 0.12;
        ELSIF Velocity_SPms >= 0.0 THEN 
            PosRef := Velocity_SPms;
        ELSE 
            PosRef := 0.0;
        END_IF;

        (* End of Saturate: '<S3>/Saturation2' *)
        

        (* MATLAB Function: '<S3>/RampSignal' *)
        (* MATLAB Function 'Subsystem/RampMotionProfileGenerator/RampSignal': '<S5>:1' *)
        (* '<S5>:1:2' x_SP = x_ref - x0; *)
        (* '<S5>:1:3' vs=v_ref; *)
        (* '<S5>:1:4' slopeExt=v0-vs; *)
        (* '<S5>:1:5' slopeRetr=-vs-v0; *)
        (* '<S5>:1:7' as = vs/tRamp; *)
        (* '<S5>:1:8' s_acc=(vs^2-v0^2)/as; *)
        (* '<S5>:1:10' tHold=(x_SP-s_acc)/vs; *)
        tHold := ((rtb_Saturation3 - x0m) - (((PosRef * PosRef) - (v0ms * v0ms)) / (PosRef / tRamps))) / PosRef;
        (* '<S5>:1:12' if tHold < 0 *)

        IF tHold < 0.0 THEN 
            (* '<S5>:1:13' Error = 1; *)
            Error := 1;
        ELSE 
            (* '<S5>:1:14' else *)
            (* '<S5>:1:15' Error = 0; *)
            Error := 0;
        END_IF;

        (* '<S5>:1:18' t1=tRamp; *)
        (* '<S5>:1:19' t2=tHold; *)
        (* '<S5>:1:20' t3=tRamp; *)
        (* '<S5>:1:21' t4=tWait; *)
        (* '<S5>:1:22' t5=t1; *)
        (* '<S5>:1:23' t6=t2; *)
        (* '<S5>:1:24' t7=t3; *)
        (* '<S5>:1:26' x1 = x0 + v0*((t0+t1)-t0)-(slopeExt/t1)*((t0+t1)-t0)^2/2; *)
        a_tmp_tmp := t0s + tRamps;
        a_tmp := a_tmp_tmp - t0s;
        x1_tmp := (v0ms - PosRef) / tRamps;
        x1 := ((a_tmp * v0ms) + x0m) - ((x1_tmp * (a_tmp * a_tmp)) / 2.0);
        (* '<S5>:1:27' x2 = x1 + vs*((t0+t1+t2)-(t0+t1)); *)
        (* '<S5>:1:28' x4 = x_ref - v0*((t0+t1+t2+t3+t4+t5)-(t0+t1+t2+t3+t4))+(slopeRetr/t5)*((t0+t1+t2+t3+t4+t5)-(t0+t1+t2+t3+t4))^2/2; *)
        a_tmp_tmp_0 := a_tmp_tmp + tHold;
        a_tmp_tmp_1 := a_tmp_tmp_0 + tRamps;
        a_tmp := a_tmp_tmp_1 + tHoldPoss;
        a_tmp_tmp_2 := a_tmp + tRamps;
        a_tmp_0 := a_tmp_tmp_2 - a_tmp;
        x4_tmp := (( -PosRef) - v0ms) / tRamps;
        x4 := (rtb_Saturation3 - (a_tmp_0 * v0ms)) + ((x4_tmp * (a_tmp_0 * a_tmp_0)) / 2.0);
        (* '<S5>:1:29' x5 = x4-vs*((t0+t1+t2+t3+t4+t5+t6)-(t0+t1+t2+t3+t4+t5)); *)
        (* '<S5>:1:31' if Error == 1 *)

        IF Error = 1 THEN 
            (* '<S5>:1:32' x = x0; *)
            rtb_Saturation3 := x0m;
            (* '<S5>:1:33' v = v0; *)
            PosRef := v0ms;
        ELSIF (rtb_Time >= 0.0) AND (rtb_Time < t0s) THEN 
            (* '<S5>:1:34' elseif t>=0 && t<t0 *)
            (* '<S5>:1:35' x = x0; *)
            rtb_Saturation3 := x0m;
            (* '<S5>:1:36' v = v0; *)
            PosRef := v0ms;
        ELSIF (rtb_Time >= t0s) AND (rtb_Time < a_tmp_tmp) THEN 
            (* '<S5>:1:37' elseif t>=t0 && t<(t0+t1) *)
            (* '<S5>:1:38' x = x0 + v0*(t-t0)-(slopeExt/t1)*(t-t0)^2/2; *)
            rtb_Time := rtb_Time - t0s;
            rtb_Saturation3 := ((rtb_Time * v0ms) + x0m) - ((x1_tmp * (rtb_Time * rtb_Time)) / 2.0);
            (* '<S5>:1:39' v = v0-(slopeExt/t1)*(t-t0); *)
            PosRef := v0ms - (x1_tmp * rtb_Time);
        ELSIF (rtb_Time >= a_tmp_tmp) AND (rtb_Time < a_tmp_tmp_0) THEN 
            (* '<S5>:1:40' elseif t>=(t0+t1) && t<(t0+t1+t2) *)
            (* '<S5>:1:41' x = x1 + vs*(t-(t0+t1)); *)
            rtb_Saturation3 := ((rtb_Time - a_tmp_tmp) * PosRef) + x1;
            (* '<S5>:1:42' v = vs; *)
        ELSIF (rtb_Time >= a_tmp_tmp_0) AND (rtb_Time < a_tmp_tmp_1) THEN 
            (* '<S5>:1:43' elseif t>=(t0+t1+t2) && t<(t0+t1+t2+t3) *)
            (* '<S5>:1:44' x = x2+vs*(t-(t0+t1+t2))+(slopeExt/t3)*(t-(t0+t1+t2))^2/2; *)
            rtb_Time := rtb_Time - a_tmp_tmp_0;
            rtb_Saturation3 := ((((a_tmp_tmp_0 - a_tmp_tmp) * PosRef) + x1) + (rtb_Time * PosRef)) + ((x1_tmp * (rtb_Time * rtb_Time)) / 2.0);
            (* '<S5>:1:45' v = vs+(slopeExt/t3)*(t-(t0+t1+t2)); *)
            PosRef := (rtb_Time * x1_tmp) + PosRef;
        ELSIF (rtb_Time >= a_tmp_tmp_1) AND (rtb_Time < a_tmp) THEN 
            (* '<S5>:1:46' elseif t>=(t0+t1+t2+t3) && t<(t0+t1+t2+t3+t4) *)
            (* '<S5>:1:47' x = x_ref; *)
            (* '<S5>:1:48' v = v0; *)
            PosRef := v0ms;
        ELSIF (rtb_Time >= a_tmp) AND (rtb_Time < a_tmp_tmp_2) THEN 
            (* '<S5>:1:49' elseif t>=(t0+t1+t2+t3+t4) && t<(t0+t1+t2+t3+t4+t5) *)
            (* '<S5>:1:50' x = x_ref - v0*(t-(t0+t1+t2+t3+t4))+(slopeRetr/t5)*(t-(t0+t1+t2+t3+t4))^2/2; *)
            a_tmp := rtb_Time - a_tmp;
            rtb_Saturation3 := (rtb_Saturation3 - (a_tmp * v0ms)) + ((x4_tmp * (a_tmp * a_tmp)) / 2.0);
            (* '<S5>:1:51' v = v0+(slopeRetr/t5)*(t-(t0+t1+t2+t3+t4)); *)
            PosRef := (a_tmp * x4_tmp) + v0ms;
        ELSE 
            rtb_Saturation3 := a_tmp_tmp_2 + tHold;

            IF (rtb_Time >= a_tmp_tmp_2) AND (rtb_Time < rtb_Saturation3) THEN 
                (* '<S5>:1:52' elseif t>=(t0+t1+t2+t3+t4+t5) && t<(t0+t1+t2+t3+t4+t5+t6) *)
                (* '<S5>:1:53' x = x4-vs*(t-(t0+t1+t2+t3+t4+t5)); *)
                rtb_Saturation3 := x4 - ((rtb_Time - a_tmp_tmp_2) * PosRef);
                (* '<S5>:1:54' v = -vs; *)
                PosRef :=  -PosRef;
            ELSIF (rtb_Time >= rtb_Saturation3) AND (rtb_Time < (rtb_Saturation3 + tRamps)) THEN 
                (* '<S5>:1:55' elseif t>=(t0+t1+t2+t3+t4+t5+t6) && t<(t0+t1+t2+t3+t4+t5+t6+t7) *)
                (* '<S5>:1:56' x = x5-vs*(t-(t0+t1+t2+t3+t4+t5+t6))-(slopeRetr/t3)*(t-(t0+t1+t2+t3+t4+t5+t6))^2/2; *)
                rtb_Time := rtb_Time - rtb_Saturation3;
                rtb_Saturation3 := ((x4 - ((rtb_Saturation3 - a_tmp_tmp_2) * PosRef)) - (rtb_Time * PosRef)) - ((x4_tmp * (rtb_Time * rtb_Time)) / 2.0);
                (* '<S5>:1:57' v = -vs-(slopeRetr/t3)*(t-(t0+t1+t2+t3+t4+t5+t6)); *)
                PosRef := ( -PosRef) - (rtb_Time * x4_tmp);
            ELSE 
                (* '<S5>:1:58' else *)
                (* '<S5>:1:59' x = x0; *)
                rtb_Saturation3 := x0m;
                (* '<S5>:1:60' v = v0; *)
                PosRef := v0ms;
            END_IF;

        END_IF;

        (* End of MATLAB Function: '<S3>/RampSignal' *)
        

        (* Switch: '<S3>/Switch' *)
        (* '<S5>:1:63' T = t0+t1+t2+t3+t4+t5+t6+t7; *)

        IF  NOT Enable THEN 
            PosRef := v0ms;
        END_IF;

        (* End of Switch: '<S3>/Switch' *)
        

        (* Saturate: '<S3>/Saturation' *)

        IF PosRef > 150.0 THEN 
            (* Outport: '<Root>/VelRef' *)
            VelRef := 150.0;
        ELSIF PosRef >= -150.0 THEN 
            (* Outport: '<Root>/VelRef' *)
            VelRef := PosRef;
        ELSE 
            (* Outport: '<Root>/VelRef' *)
            VelRef := -150.0;
        END_IF;

        (* End of Saturate: '<S3>/Saturation' *)
        

        (* Switch: '<S3>/Switch1' *)

        IF Enable THEN 
            PosRef := rtb_Saturation3;
        ELSE 
            PosRef := x0m;
        END_IF;

        (* End of Switch: '<S3>/Switch1' *)
        

        (* Saturate: '<S3>/Saturation1' *)

        IF PosRef > 500.0 THEN 
            (* Outport: '<Root>/PosRef' *)
            PosRef := 500.0;
        ELSIF PosRef < 0.0 THEN 
            (* Outport: '<Root>/PosRef' *)
            PosRef := 0.0;
        END_IF;

        (* End of Saturate: '<S3>/Saturation1' *)
        (* End of Outputs for SubSystem: '<S1>/RampMotionProfileGenerator' *)
        

        (* Update for DiscreteIntegrator: '<S2>/Discrete-Time Integrator' *)
        c_DiscreteTimeIntegrator_DS := c_DiscreteTimeIntegrator_DS + 0.001;
        (* End of Outputs for SubSystem: '<Root>/Subsystem' *)
END_CASE;

END_FUNCTION_BLOCK

// ---- GlobalTextList.TcGTLO
TEXTLIST GlobalTextList
  534 = 'Actual Height: %f'
  501 = 'Actual Height: %f [m]'
  920 = 'Closed Loop Position Control ON'
  583 = 'Current Cylinder Pos: %f [m] '
  824 = 'Current Drum Pos: %f [m] '
  35 = 'Current Drum Pos: %f [°] '
  829 = 'Current I-gain: %0.1f '
  196 = 'Current MaxError: %f [m] '
  955 = 'Current MaxFlow: %0.1f [L/min] '
  137 = 'Current P-gain: %0.1f '
  907 = 'Current Position: %f [m] '
  296 = 'Current Wire Pos: %f [m] '
  628 = 'Cylinder'
  783 = 'Desired Height: %f'
  51 = 'Desired Height: %f [m]'
  854 = 'Enable Cyl'
  32 = 'Enable Winch'
  995 = 'error: %f'
  246 = 'Error: %f [mm]'
  928 = 'Error: %f [m]'
  392 = 'Feed Forward Tuning'
  423 = 'Height stabilisation'
  252 = 'Height: %f'
  904 = 'Hold Pos time: %0.1f [s] '
  81 = 'Integral Controller Gain'
  573 = 'Integral Controller ON'
  261 = 'Max Position Error'
  415 = 'Motion Reference Generator Settings'
  655 = 'New I-gain: %0.1f '
  683 = 'New MaxError: %f  [m]'
  330 = 'New MaxFlow: %0.1f [L/min] '
  347 = 'New P-gain: %0.1f '
  463 = 'Position SP: %f [m] '
  982 = 'Proportional  Controller Gain'
  215 = 'Ramp time: %0.1f [s] '
  695 = 'Set New Value'
  828 = 'Start delay: %0.1f [s] '
  775 = 'Start Height: %f [m] '
  78 = 'Start Position: %f [m] '
  983 = 'Start Velocity: %f [m/s] '
  999 = 'Velocity SP: %f [m/s] '
  560 = 'VelocityFeed Forward Controller ON'
  349 = 'Winch'
  599 = 'Zero offset: %f '
  396 = 'Zero offset: %f [m]'
  522 = 'Zero offset: %f [m] '
END_TEXTLIST

// ---- HMI/Main.TcVIS
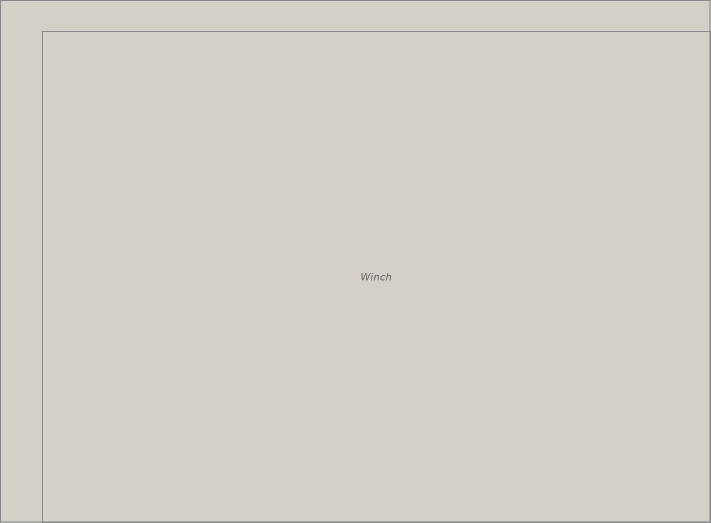
VISUALIZATION Main  // 711x523
    TabControl (42,31 669x492)
        shows Winch()
        shows Cylinder()
        [0]: TabTitle=Winch
        [1]: TabTitle=Cylinder
END_VISUALIZATION

// ---- HMI/Sub/Cylinder.TcVIS
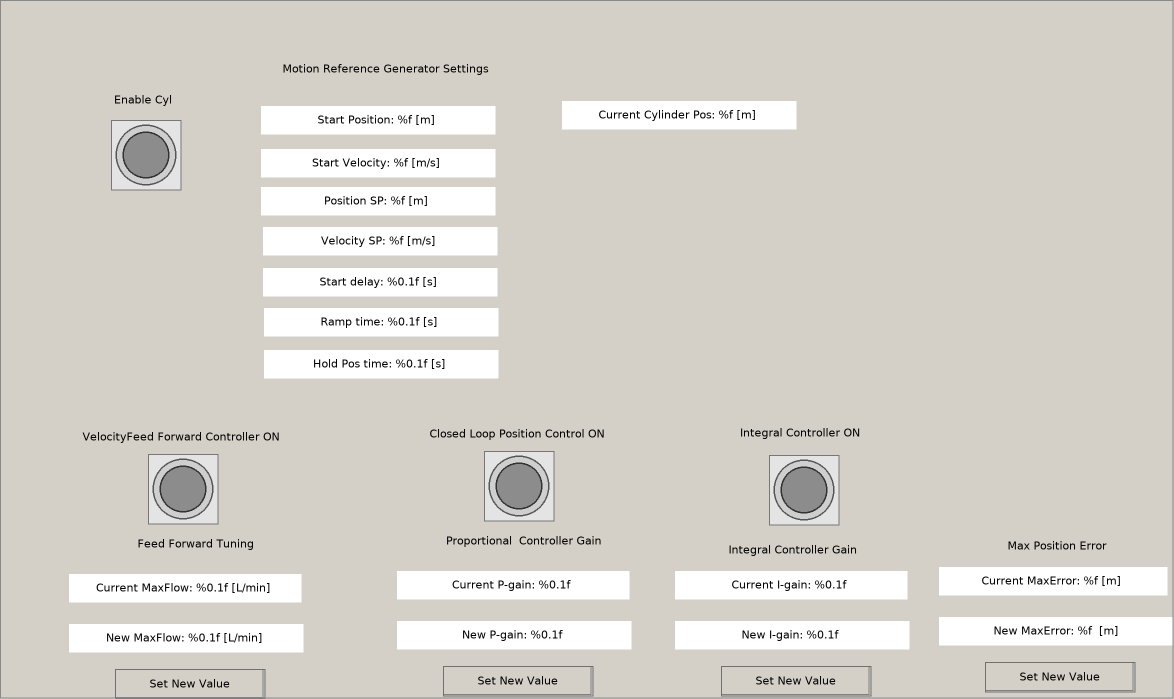
VISUALIZATION Cylinder  // 1174x699
    Label (68,85 150x30), "Enable Cyl"
    PushSwitch (111,120 70x70), variable: G_Hmi.bCylEnable, behaviour: TOGGLE, style: Switch-PushSwitch-Gray
    Label (240,54 291x30), "Motion Reference Generator Settings"
    Textfield (260,105 236x30), "Start Position: %f [m]", text variable: G_Hmi.stMotionReferenceGeneratorSettingsCylinder.fStartPosition_m
        OnMouseDown: write the text variable via Default, min 0, max 0.5
    Textfield (260,148 236x30), "Start Velocity: %f [m/s]", text variable: G_Hmi.stMotionReferenceGeneratorSettingsCylinder.fStartVelocity_m
        OnMouseDown: write the text variable via Default, min 0, max 0.05
    Textfield (260,186 236x30), "Position SP: %f [m]", text variable: G_Hmi.stMotionReferenceGeneratorSettingsCylinder.fPositionSetpoint_ms
        OnMouseDown: write the text variable via Default, min 0, max 0.45
    Textfield (262,226 236x30), "Velocity SP: %f [m/s]", text variable: G_Hmi.stMotionReferenceGeneratorSettingsCylinder.fVelocitySetpoint_m
        OnMouseDown: write the text variable via Default, min 0, max 0.05
    Textfield (262,267 236x30), "Start delay: %0.1f [s]", text variable: G_Hmi.stMotionReferenceGeneratorSettingsCylinder.fTimeBeforeStarting_s
        OnMouseDown: write the text variable via Default, min 0, max 10
    Textfield (263,307 236x30), "Ramp time: %0.1f [s]", text variable: G_Hmi.stMotionReferenceGeneratorSettingsCylinder.fRampTime_s
        OnMouseDown: write the text variable via Default, min 0, max 10
    Textfield (263,349 236x30), "Hold Pos time: %0.1f [s]", text variable: G_Hmi.stMotionReferenceGeneratorSettingsCylinder.fHoldPositionTime_s
        OnMouseDown: write the text variable via Default, min 0, max 10
    Textfield (561,100 236x30), "Current Cylinder Pos: %f [m]", text variable: G_Sensors.fPositionCylPiston
        OnMouseDown: write the text variable via Default, min 0, max 0.5
    Button (443,666 150x30), "Set New Value"
        tap G_Hmi.stModifyAutomaticControlSettingsCylinder.bSetNewProportionalGain
    Textfield (396,570 234x30), "Current P-gain: %0.1f", text variable: G_Parameters.stParam.stClosedLoopControlSettingsCylinder.fProportionalGain
    Textfield (396,620 236x30), "New P-gain: %0.1f", text variable: G_Hmi.stModifyAutomaticControlSettingsCylinder.fNewProportionalGain
        OnMouseDown: write the text variable via Default
    Label (441,526 166x30), "Proportional Controller Gain"
    Button (721,666 150x30), "Set New Value"
        tap G_Hmi.stModifyAutomaticControlSettingsCylinder.bSetNewIntegralGain
    Textfield (674,570 234x30), "Current I-gain: %0.1f", text variable: G_Parameters.stParam.stClosedLoopControlSettingsCylinder.fIntegralGain
    Textfield (674,620 236x30), "New I-gain: %0.1f", text variable: G_Hmi.stModifyAutomaticControlSettingsCylinder.fNewIntegralGain
        OnMouseDown: write the text variable via Default
    Label (718,535 150x30), "Integral Controller Gain"
    PushSwitch (769,455 70x70), variable: G_Hmi.stAutomaticControlSettingsCylinder.bEnableIntegralController, behaviour: TOGGLE, style: Switch-PushSwitch-Gray
    Label (717,418 166x30), "Integral Controller ON"
    Label (391,419 252x30), "Closed Loop Position Control ON"
    PushSwitch (484,451 70x70), variable: G_Hmi.stAutomaticControlSettingsCylinder.bEnableClosedLoopPositionControl, behaviour: TOGGLE, style: Switch-PushSwitch-Gray
    Label (55,422 252x30), "VelocityFeed Forward Controller ON"
    PushSwitch (148,454 70x70), variable: G_Hmi.stAutomaticControlSettingsCylinder.bEnableVelocityFeedForwardControl, behaviour: TOGGLE, style: Switch-PushSwitch-Gray
    Button (115,669 150x30), "Set New Value"
        tap G_Hmi.stModifyAutomaticControlSettingsCylinder.bSetNewMaxFlowCapacity p1329445385=TRUE
    Textfield (68,573 234x30), "Current MaxFlow: %0.1f [L/min]", text variable: G_Parameters.stParam.stOpenLoopControlSettingsCylinder.fMaxFlowCapacity
    Textfield (68,623 236x30), "New MaxFlow: %0.1f [L/min]", text variable: G_Hmi.stModifyAutomaticControlSettingsCylinder.fNewMaxFlowCapacity
        OnMouseDown: write the text variable via Default, min 0.0001, max 100
    Label (113,529 166x30), "Feed Forward Tuning"
    Button (985,662 150x30), "Set New Value"
        tap G_Hmi.stModifyAutomaticControlSettingsCylinder.bSetNewMaxPositionError
    Textfield (938,566 230x30), "Current MaxError: %f [m]", text variable: G_Parameters.stParam.stClosedLoopControlSettingsCylinder.fMaxPositionError
    Textfield (938,616 236x30), "New MaxError: %f [m]", text variable: G_Hmi.stModifyAutomaticControlSettingsCylinder.fNewMaxPositionError
        OnMouseDown: write the text variable via Default
    Label (982,531 150x30), "Max Position Error"
END_VISUALIZATION

// ---- HMI/Sub/Winch.TcVIS
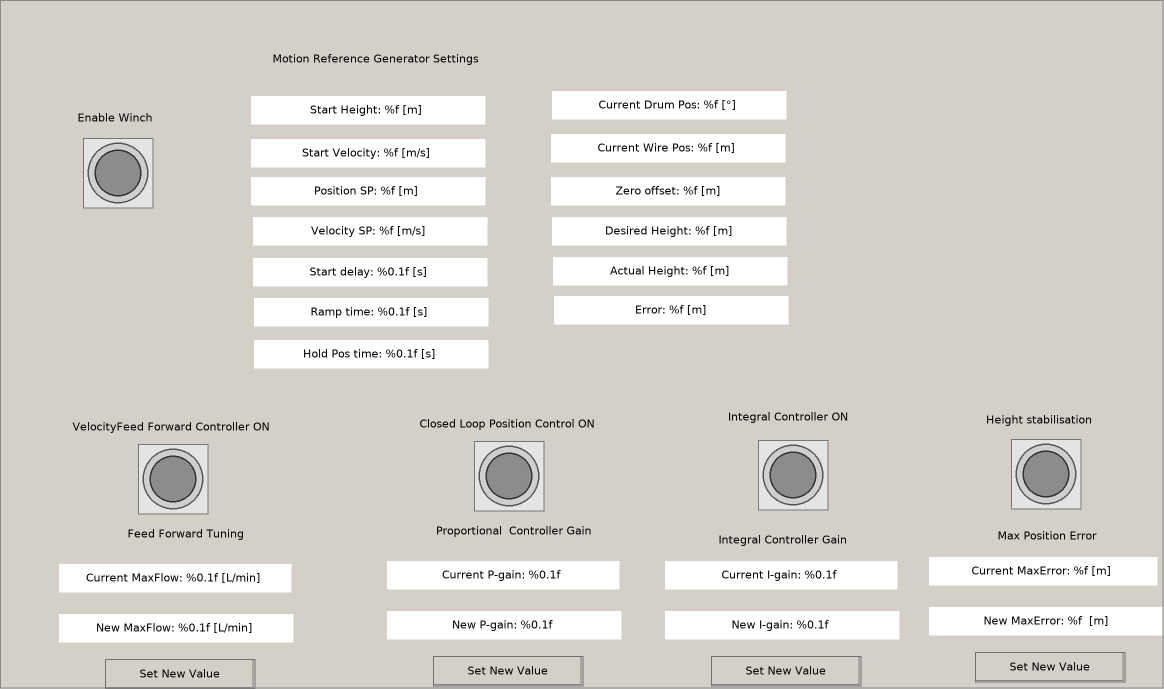
VISUALIZATION Winch  // 1164x689
    Label (40,103 150x30), "Enable Winch"
    PushSwitch (83,138 70x70), variable: G_Hmi.bWinchEnable, behaviour: TOGGLE, style: Switch-PushSwitch-Gray
    Label (230,44 291x30), "Motion Reference Generator Settings"
    Textfield (250,95 236x30), "Start Height: %f [m]", text variable: G_Hmi.stMotionReferenceGeneratorSettingsWinch.fStartPosition_m
        OnMouseDown: write the text variable via Default, min 0, max 1.0
    Textfield (250,138 236x30), "Start Velocity: %f [m/s]", text variable: G_Hmi.stMotionReferenceGeneratorSettingsWinch.fStartVelocity_m
        OnMouseDown: write the text variable via Default, min 0, max 0.05
    Textfield (250,176 236x30), "Position SP: %f [m]", text variable: G_Hmi.stMotionReferenceGeneratorSettingsWinch.fPositionSetpoint_ms
        OnMouseDown: write the text variable via Default, min 0, max 1.0
    Textfield (252,216 236x30), "Velocity SP: %f [m/s]", text variable: G_Hmi.stMotionReferenceGeneratorSettingsWinch.fVelocitySetpoint_m
        OnMouseDown: write the text variable via Default, min 0, max 0.05
    Textfield (252,257 236x30), "Start delay: %0.1f [s]", text variable: G_Hmi.stMotionReferenceGeneratorSettingsWinch.fTimeBeforeStarting_s
        OnMouseDown: write the text variable via Default, min 0, max 10
    Textfield (253,297 236x30), "Ramp time: %0.1f [s]", text variable: G_Hmi.stMotionReferenceGeneratorSettingsWinch.fRampTime_s
        OnMouseDown: write the text variable via Default, min 0, max 10
    Textfield (253,339 236x30), "Hold Pos time: %0.1f [s]", text variable: G_Hmi.stMotionReferenceGeneratorSettingsWinch.fHoldPositionTime_s
        OnMouseDown: write the text variable via Default, min 0, max 10
    Textfield (551,90 236x30), "Current Drum Pos: %f [°]", text variable: G_Sensors.fWinchEncoderPosition
        OnMouseDown: write the text variable via Default, min 0, max 0.5
    Button (433,656 150x30), "Set New Value"
        tap G_Hmi.stModifyAutomaticControlSettingsWinch.bSetNewProportionalGain
    Textfield (386,560 234x30), "Current P-gain: %0.1f", text variable: G_Parameters.stParam.stClosedLoopControlSettingsWinch.fProportionalGain
    Textfield (386,610 236x30), "New P-gain: %0.1f", text variable: G_Hmi.stModifyAutomaticControlSettingsWinch.fNewProportionalGain
        OnMouseDown: write the text variable via Default
    Label (431,516 166x30), "Proportional Controller Gain"
    Button (711,656 150x30), "Set New Value"
        tap G_Hmi.stModifyAutomaticControlSettingsWinch.bSetNewIntegralGain
    Textfield (664,560 234x30), "Current I-gain: %0.1f", text variable: G_Parameters.stParam.stClosedLoopControlSettingsWinch.fIntegralGain
    Textfield (664,610 236x30), "New I-gain: %0.1f", text variable: G_Hmi.stModifyAutomaticControlSettingsWinch.fNewIntegralGain
        OnMouseDown: write the text variable via Default
    Label (708,525 150x30), "Integral Controller Gain"
    PushSwitch (758,440 70x70), variable: G_Hmi.stAutomaticControlSettingsWinch.bEnableIntegralController, behaviour: TOGGLE, style: Switch-PushSwitch-Gray
    Label (705,402 166x30), "Integral Controller ON"
    Label (381,409 252x30), "Closed Loop Position Control ON"
    PushSwitch (474,441 70x70), variable: G_Hmi.stAutomaticControlSettingsWinch.bEnableClosedLoopPositionControl, behaviour: TOGGLE, style: Switch-PushSwitch-Gray
    Label (45,412 252x30), "VelocityFeed Forward Controller ON"
    PushSwitch (138,444 70x70), variable: G_Hmi.stAutomaticControlSettingsWinch.bEnableVelocityFeedForwardControl, behaviour: TOGGLE, style: Switch-PushSwitch-Gray
    Button (105,659 150x30), "Set New Value"
        tap G_Hmi.stModifyAutomaticControlSettingsWinch.bSetNewMaxFlowCapacity p1329445385=TRUE
    Textfield (58,563 234x30), "Current MaxFlow: %0.1f [L/min]", text variable: G_Parameters.stParam.stOpenLoopControlSettingsWinch.fMaxFlowCapacity
    Textfield (58,613 236x30), "New MaxFlow: %0.1f [L/min]", text variable: G_Hmi.stModifyAutomaticControlSettingsWinch.fNewMaxFlowCapacity
        OnMouseDown: write the text variable via Default, min 0.0001, max 100
    Label (103,519 166x30), "Feed Forward Tuning"
    Button (975,652 150x30), "Set New Value"
        tap G_Hmi.stModifyAutomaticControlSettingsWinch.bSetNewMaxPositionError
    Textfield (928,556 230x30), "Current MaxError: %f [m]", text variable: G_Parameters.stParam.stClosedLoopControlSettingsWinch.fMaxPositionError
    Textfield (928,606 236x30), "New MaxError: %f [m]", text variable: G_Hmi.stModifyAutomaticControlSettingsWinch.fNewMaxPositionError
        OnMouseDown: write the text variable via Default
    Label (972,521 150x30), "Max Position Error"
    Textfield (550,133 236x30), "Current Wire Pos: %f [m]", text variable: G_Sensors.fWinchWirePosition
        OnMouseDown: write the text variable via Default, min 0, max 0.5
    PushSwitch (1011,439 70x70), variable: G_HeightCorrection.xCorrectHeight, behaviour: TOGGLE, style: Switch-PushSwitch-Gray
    Label (956,405 166x30), "Height stabilisation"
    Textfield (550,176 236x30), "Zero offset: %f [m]", text variable: G_HeightCorrection.rZeroOffset
        OnMouseDown: write the text variable via Default, min -100.0, max 100.0
    Textfield (551,216 236x30), "Desired Height: %f [m]", text variable: G_HeightCorrection.rDesiredHeight
        OnMouseDown: write the text variable via Default, min 0, max 0.5
    Textfield (552,256 236x30), "Actual Height: %f [m]", text variable: G_HeightCorrection.rActual
        OnMouseDown: write the text variable via Default, min 0, max 0.5
    Textfield (553,295 236x30), "Error: %f [m]", text variable: G_Sensors.fWinchWirePosition
        OnMouseDown: write the text variable via Default, min 0, max 0.5
END_VISUALIZATION
